C05373=1017.378,25.975,-122.265,-24.216,21.496,-42.540
C05374=1017.376,26.375,-122.301,-24.217,21.496,-42.534
C05375=1017.374,26.774,-122.336,-24.218,21.495,-42.529
C05376=1017.373,27.173,-122.371,-24.218,21.494,-42.525
C05377=1017.372,27.573,-122.406,-24.219,21.495,-42.520
C05378=1017.370,27.972,-122.441,-24.219,21.493,-42.516
C05379=1017.368,28.372,-122.475,-24.220,21.493,-42.510
C05380=1017.366,28.772,-122.511,-24.221,21.493,-42.507
C05381=1017.364,29.171,-122.546,-24.221,21.492,-42.501
C05382=1017.363,29.570,-122.580,-24.222,21.492,-42.497
C05383=1017.360,29.970,-122.616,-24.223,21.492,-42.492
C05384=1017.358,30.370,-122.650,-24.223,21.491,-42.488
C05385=1017.357,30.769,-122.685,-24.224,21.491,-42.483
C05386=1017.354,31.168,-122.721,-24.224,21.490,-42.479
C05387=1017.354,31.568,-122.756,-24.225,21.490,-42.474
C05388=1017.351,31.968,-122.791,-24.226,21.489,-42.469
C05389=1017.349,32.368,-122.826,-24.226,21.489,-42.464
C05390=1017.347,32.767,-122.861,-24.227,21.489,-42.461
C05391=1017.345,33.166,-122.896,-24.228,21.489,-42.455
C05392=1017.344,33.567,-122.932,-24.228,21.487,-42.451
C05393=1017.341,33.966,-122.968,-24.229,21.488,-42.446
C05394=1017.339,34.366,-123.002,-24.229,21.487,-42.442
C05395=1017.337,34.766,-123.037,-24.230,21.486,-42.437
C05396=1017.335,35.165,-123.073,-24.231,21.486,-42.433
C05397=1017.334,35.565,-123.108,-24.231,21.486,-42.428
C05398=1017.331,35.965,-123.143,-24.232,21.486,-42.424
C05399=1017.329,36.365,-123.178,-24.233,21.485,-42.418
C05400=1017.327,36.764,-123.214,-24.233,21.484,-42.414
C05401=1017.325,37.164,-123.250,-24.234,21.485,-42.409
C05402=1017.323,37.564,-123.284,-24.235,21.484,-42.405
C05403=1017.321,37.964,-123.320,-24.235,21.483,-42.400
C05404=1017.318,38.363,-123.355,-24.236,21.483,-42.396
C05405=1017.316,38.764,-123.391,-24.237,21.483,-42.391
C05406=1017.314,39.164,-123.426,-24.237,21.483,-42.387
C05407=1017.312,39.563,-123.461,-24.238,21.482,-42.383
C05408=1017.310,39.964,-123.497,-24.238,21.481,-42.378
C05409=1017.307,40.363,-123.533,-24.239,21.481,-42.374
C05410=1017.305,40.763,-123.568,-24.240,21.481,-42.369
C05411=1017.303,41.164,-123.603,-24.240,21.481,-42.365
C05412=1017.301,41.563,-123.639,-24.241,21.480,-42.359
C05413=1017.297,41.964,-123.674,-24.241,21.479,-42.356
C05414=1017.295,42.363,-123.710,-24.242,21.479,-42.352
C05415=1017.293,42.763,-123.746,-24.243,21.479,-42.347
C05416=1017.291,43.163,-123.781,-24.243,21.479,-42.343
C05417=1017.288,43.563,-123.816,-24.244,21.479,-42.338
C05418=1017.286,43.964,-123.853,-24.244,21.477,-42.333
C05419=1017.284,44.363,-123.888,-24.245,21.477,-42.330
C05420=1017.281,44.763,-123.924,-24.246,21.477,-42.325
C05421=1017.279,45.164,-123.959,-24.246,21.477,-42.321
C05422=1017.276,45.563,-123.995,-24.247,21.477,-42.316
C05423=1017.274,45.964,-124.031,-24.247,21.475,-42.311
C05424=1017.271,46.363,-124.067,-24.248,21.475,-42.308
C05425=1017.269,46.764,-124.102,-24.249,21.475,-42.302
C05426=1017.266,47.164,-124.138,-24.249,21.475,-42.299
C05427=1017.264,47.564,-124.174,-24.250,21.474,-42.295
C05428=1017.261,47.964,-124.210,-24.251,21.474,-42.290
C05429=1017.259,48.364,-124.245,-24.251,21.474,-42.286
C05430=1017.256,48.764,-124.281,-24.251,21.472,-42.282
C05431=1017.253,49.164,-124.317,-24.252,21.473,-42.277
C05432=1017.251,49.565,-124.353,-24.253,21.472,-42.273
C05433=1017.248,49.965,-124.389,-24.254,21.472,-42.268
C05434=1017.245,50.364,-124.424,-24.254,21.472,-42.264
C05435=1017.243,50.765,-124.461,-24.255,21.471,-42.260
C05436=1017.239,51.165,-124.496,-24.255,21.471,-42.255
C05437=1017.237,51.565,-124.532,-24.256,21.471,-42.251
C05438=1017.235,51.965,-124.568,-24.256,21.470,-42.247
C05439=1017.232,52.365,-124.604,-24.257,21.469,-42.243
C05440=1017.229,52.765,-124.640,-24.258,21.469,-42.238
C05441=1017.227,53.166,-124.675,-24.258,21.469,-42.234
C05442=1017.223,53.566,-124.712,-24.259,21.468,-42.230
C05443=1017.220,53.966,-124.748,-24.259,21.468,-42.225
C05444=1017.218,54.366,-124.784,-24.260,21.468,-42.221
C05445=1017.215,54.767,-124.820,-24.260,21.468,-42.218
C05446=1017.211,55.167,-124.856,-24.261,21.468,-42.212
C05447=1017.209,55.567,-124.892,-24.262,21.467,-42.209
C05448=1017.206,55.967,-124.928,-24.262,21.467,-42.205
C05449=1017.203,56.367,-124.964,-24.263,21.465,-42.201
C05450=1017.200,56.768,-125.000,-24.264,21.466,-42.196
C05451=1017.197,57.168,-125.036,-24.264,21.465,-42.192
C05452=1017.194,57.568,-125.072,-24.264,21.465,-42.188
C05453=1017.192,57.968,-125.109,-24.265,21.465,-42.183
C05454=1017.188,58.368,-125.145,-24.266,21.464,-42.179
C05455=1017.185,58.769,-125.180,-24.266,21.464,-42.175
C05456=1017.182,59.168,-125.217,-24.267,21.463,-42.172
C05457=1017.180,59.569,-125.253,-24.268,21.464,-42.166
C05458=1017.176,59.969,-125.289,-24.268,21.463,-42.163
C05459=1017.173,60.369,-125.325,-24.269,21.463,-42.159
C05460=1017.170,60.769,-125.361,-24.269,21.462,-42.155
C05461=1017.167,61.169,-125.399,-24.270,21.462,-42.150
C05462=1017.164,61.570,-125.434,-24.270,21.462,-42.146
C05463=1017.161,61.970,-125.470,-24.271,21.461,-42.142
C05464=1017.158,62.370,-125.506,-24.271,21.461,-42.139
C05465=1017.154,62.790,-125.545,-24.272,21.460,-42.133
C05466=1017.153,63.043,-125.568,-24.272,21.460,-42.131
C05467=1017.150,63.311,-125.593,-24.273,21.460,-42.129
C05468=1017.148,63.561,-125.615,-24.273,21.459,-42.127
C05469=1017.146,63.777,-125.634,-24.274,21.460,-42.124
C05470=1017.144,63.984,-125.653,-24.274,21.460,-42.122
C05471=1017.143,64.202,-125.673,-24.274,21.459,-42.120
C05472=1017.141,64.431,-125.693,-24.274,21.459,-42.116
C05473=1017.139,64.668,-125.715,-24.275,21.459,-42.115
C05474=1017.138,64.903,-125.737,-24.275,21.458,-42.113
C05475=1017.135,65.133,-125.758,-24.275,21.458,-42.111
C05476=1017.134,65.355,-125.778,-24.276,21.459,-42.108
C05477=1017.131,65.568,-125.797,-24.276,21.458,-42.106
C05478=1017.128,65.975,-125.834,-24.277,21.458,-42.102
C05479=1017.125,66.374,-125.870,-24.277,21.457,-42.098
C05480=1017.121,66.774,-125.907,-24.278,21.457,-42.094
C05481=1017.118,67.177,-125.943,-24.278,21.457,-42.089
C05482=1017.115,67.581,-125.980,-24.279,21.457,-42.085
C05483=1017.111,67.985,-126.017,-24.279,21.456,-42.082
C05484=1017.109,68.391,-126.053,-24.280,21.456,-42.078
C05485=1017.104,68.798,-126.091,-24.280,21.455,-42.074
C05486=1017.101,69.207,-126.128,-24.281,21.455,-42.069
C05487=1017.098,69.617,-126.166,-24.282,21.455,-42.065
C05488=1017.094,70.028,-126.204,-24.282,21.454,-42.061
C05489=1017.090,70.440,-126.241,-24.283,21.454,-42.058
C05490=1017.087,70.850,-126.278,-24.283,21.453,-42.054
C05491=1017.083,71.261,-126.316,-24.284,21.454,-42.049
C05492=1017.079,71.673,-126.353,-24.285,21.453,-42.045
C05493=1017.076,72.084,-126.391,-24.285,21.453,-42.041
C05494=1017.072,72.498,-126.429,-24.285,21.452,-42.037
C05495=1017.069,72.913,-126.467,-24.286,21.452,-42.034
C05496=1017.064,73.331,-126.505,-24.287,21.452,-42.028
C05497=1017.061,73.752,-126.543,-24.287,21.452,-42.025
C05498=1017.059,73.963,-126.563,-24.288,21.451,-42.023
C05499=1017.057,74.175,-126.582,-24.288,21.451,-42.021
C05500=1017.055,74.388,-126.602,-24.288,21.451,-42.019
C05501=1017.054,74.601,-126.621,-24.288,21.451,-42.017
C05502=1017.051,74.815,-126.641,-24.289,21.450,-42.015
C05503=1017.050,75.028,-126.660,-24.289,21.451,-42.012
C05504=1017.047,75.242,-126.680,-24.289,21.451,-42.010
C05505=1017.045,75.454,-126.699,-24.290,21.450,-42.008
C05506=1017.041,75.873,-126.738,-24.290,21.450,-42.004
C05507=1017.037,76.286,-126.776,-24.291,21.449,-42.001
C05508=1017.034,76.687,-126.812,-24.291,21.449,-41.997
C05509=1017.030,77.082,-126.848,-24.292,21.449,-41.994
C05510=1017.026,77.471,-126.885,-24.292,21.448,-41.989
C05511=1017.023,77.856,-126.919,-24.293,21.447,-41.986
C05512=1017.019,78.243,-126.954,-24.293,21.448,-41.980
C05513=1017.015,78.634,-126.991,-24.294,21.447,-41.977
C05514=1017.011,79.031,-127.028,-24.294,21.447,-41.973
C05515=1017.008,79.436,-127.065,-24.295,21.447,-41.970
C05516=1017.004,79.850,-127.103,-24.296,21.447,-41.966
C05517=1017.001,80.061,-127.122,-24.296,21.446,-41.964
C05518=1016.999,80.273,-127.141,-24.296,21.446,-41.962
C05519=1016.997,80.485,-127.161,-24.296,21.446,-41.960
C05520=1016.995,80.698,-127.180,-24.297,21.446,-41.958
C05521=1016.993,80.911,-127.200,-24.297,21.445,-41.956
C05522=1016.991,81.124,-127.220,-24.297,21.445,-41.955
C05523=1016.989,81.336,-127.239,-24.297,21.445,-41.953
C05524=1016.986,81.549,-127.259,-24.298,21.445,-41.951
C05525=1016.984,81.760,-127.278,-24.298,21.445,-41.949
C05526=1016.982,81.972,-127.298,-24.298,21.444,-41.947
C05527=1016.980,82.184,-127.317,-24.299,21.445,-41.944
C05528=1016.979,82.395,-127.337,-24.299,21.444,-41.942
C05529=1016.976,82.606,-127.356,-24.299,21.444,-41.940
C05530=1016.973,82.816,-127.376,-24.299,21.444,-41.938
C05531=1016.970,83.236,-127.414,-24.300,21.444,-41.935
C05532=1016.965,83.656,-127.453,-24.300,21.444,-41.931
C05533=1016.961,84.072,-127.492,-24.301,21.443,-41.927
C05534=1016.957,84.488,-127.530,-24.301,21.443,-41.923
C05535=1016.953,84.902,-127.568,-24.302,21.443,-41.920
C05536=1016.949,85.315,-127.606,-24.302,21.442,-41.916
C05537=1016.944,85.726,-127.644,-24.303,21.442,-41.912
C05538=1016.940,86.135,-127.682,-24.303,21.441,-41.908
C05539=1016.935,86.542,-127.719,-24.304,21.442,-41.905
C05540=1016.931,86.948,-127.756,-24.304,21.441,-41.901
C05541=1016.927,87.350,-127.794,-24.305,21.441,-41.898
C05542=1016.923,87.747,-127.831,-24.305,21.440,-41.894
C05543=1016.919,88.135,-127.867,-24.306,21.440,-41.890
C05544=1016.914,88.518,-127.902,-24.307,21.440,-41.887
C05545=1016.910,88.901,-127.937,-24.307,21.440,-41.883
C05546=1016.907,89.288,-127.973,-24.308,21.439,-41.879
C05547=1016.903,89.681,-128.010,-24.308,21.439,-41.875
C05548=1016.898,90.079,-128.046,-24.309,21.439,-41.872
C05549=1016.894,90.478,-128.083,-24.309,21.439,-41.868
C05550=1016.890,90.877,-128.120,-24.310,21.438,-41.865
C05551=1016.884,91.277,-128.157,-24.310,21.438,-41.861
C05552=1016.880,91.675,-128.194,-24.311,21.438,-41.857
C05553=1016.876,92.074,-128.231,-24.311,21.438,-41.854
C05554=1016.872,92.474,-128.268,-24.312,21.437,-41.850
C05555=1016.867,92.873,-128.305,-24.312,21.437,-41.846
C05556=1016.863,93.272,-128.342,-24.312,21.437,-41.844
C05557=1016.859,93.671,-128.379,-24.313,21.436,-41.841
C05558=1016.854,94.070,-128.416,-24.313,21.436,-41.837
C05559=1016.850,94.469,-128.454,-24.314,21.435,-41.833
C05560=1016.845,94.867,-128.490,-24.315,21.436,-41.830
C05561=1016.840,95.266,-128.528,-24.315,21.435,-41.826
C05562=1016.836,95.666,-128.564,-24.316,21.435,-41.822
C05563=1016.832,96.065,-128.601,-24.316,21.435,-41.819
C05564=1016.827,96.464,-128.639,-24.317,21.435,-41.815
C05565=1016.822,96.862,-128.676,-24.317,21.434,-41.811
C05566=1016.817,97.261,-128.713,-24.318,21.434,-41.808
C05567=1016.813,97.660,-128.750,-24.318,21.433,-41.806
C05568=1016.809,98.059,-128.787,-24.318,21.433,-41.802
C05569=1016.803,98.458,-128.824,-24.319,21.432,-41.798
C05570=1016.799,98.856,-128.861,-24.319,21.433,-41.795
C05571=1016.794,99.256,-128.899,-24.320,21.432,-41.791
C05572=1016.790,99.654,-128.935,-24.320,21.432,-41.787
C05573=1016.785,100.053,-128.973,-24.321,21.432,-41.784
C05574=1016.780,100.452,-129.009,-24.322,21.432,-41.780
C05575=1016.775,100.851,-129.047,-24.322,21.431,-41.778
C05576=1016.770,101.249,-129.083,-24.322,21.431,-41.775
C05577=1016.765,101.648,-129.121,-24.323,21.431,-41.771
C05578=1016.761,102.047,-129.159,-24.323,21.430,-41.767
C05579=1016.756,102.445,-129.195,-24.324,21.430,-41.763
C05580=1016.751,102.844,-129.233,-24.324,21.430,-41.760
C05581=1016.746,103.242,-129.270,-24.325,21.430,-41.756
C05582=1016.741,103.641,-129.307,-24.325,21.430,-41.754
C05583=1016.736,104.040,-129.345,-24.326,21.429,-41.751
C05584=1016.731,104.438,-129.381,-24.326,21.429,-41.747
C05585=1016.727,104.837,-129.419,-24.327,21.429,-41.743
C05586=1016.721,105.236,-129.456,-24.327,21.429,-41.740
C05587=1016.717,105.635,-129.493,-24.328,21.428,-41.736
C05588=1016.712,106.033,-129.531,-24.328,21.428,-41.734
C05589=1016.706,106.431,-129.568,-24.328,21.427,-41.730
C05590=1016.701,106.831,-129.606,-24.329,21.427,-41.727
C05591=1016.697,107.229,-129.642,-24.330,21.427,-41.723
C05592=1016.691,107.627,-129.680,-24.330,21.427,-41.719
C05593=1016.686,108.026,-129.717,-24.330,21.426,-41.717
C05594=1016.681,108.425,-129.755,-24.331,21.426,-41.714
C05595=1016.676,108.823,-129.791,-24.331,21.426,-41.710
C05596=1016.671,109.221,-129.829,-24.332,21.426,-41.707
C05597=1016.666,109.620,-129.866,-24.332,21.426,-41.703
C05598=1016.661,110.019,-129.904,-24.333,21.425,-41.701
C05599=1016.655,110.417,-129.941,-24.333,21.425,-41.697
C05600=1016.650,110.816,-129.978,-24.334,21.425,-41.694
C05601=1016.645,111.215,-130.016,-24.334,21.425,-41.690
C05602=1016.639,111.613,-130.053,-24.334,21.424,-41.688
C05603=1016.634,112.012,-130.090,-24.335,21.423,-41.684
C05604=1016.629,112.410,-130.128,-24.335,21.424,-41.681
C05605=1016.624,112.808,-130.164,-24.336,21.423,-41.677
C05606=1016.618,113.207,-130.202,-24.336,21.423,-41.675
C05607=1016.614,113.606,-130.239,-24.337,21.423,-41.671
C05608=1016.608,114.004,-130.277,-24.337,21.422,-41.668
C05609=1016.602,114.403,-130.315,-24.338,21.423,-41.664
C05610=1016.597,114.801,-130.352,-24.338,21.422,-41.662
C05611=1016.591,115.200,-130.389,-24.339,21.422,-41.659
C05612=1016.586,115.598,-130.426,-24.339,21.422,-41.655
C05613=1016.580,115.997,-130.464,-24.340,21.422,-41.652
C05614=1016.575,116.395,-130.501,-24.340,21.421,-41.649
C05615=1016.570,116.787,-130.539,-24.340,21.420,-41.646
C05616=1016.564,117.192,-130.576,-24.341,21.421,-41.642
C05617=1016.559,117.590,-130.613,-24.341,21.420,-41.638
C05618=1016.552,117.989,-130.651,-24.342,21.420,-41.637
C05619=1016.547,118.387,-130.688,-24.342,21.420,-41.633
C05620=1016.541,118.786,-130.725,-24.343,21.420,-41.629
C05621=1016.536,119.184,-130.763,-24.343,21.420,-41.626
C05622=1016.531,119.582,-130.801,-24.343,21.419,-41.624
C05623=1016.525,119.981,-130.839,-24.344,21.419,-41.620
C05624=1016.519,120.379,-130.876,-24.345,21.419,-41.617
C05625=1016.514,120.778,-130.913,-24.345,21.418,-41.614
C05626=1016.509,121.177,-130.951,-24.345,21.418,-41.611
C05627=1016.503,121.575,-130.989,-24.346,21.418,-41.607
C05628=1016.498,121.973,-131.027,-24.346,21.417,-41.605
C05629=1016.493,122.373,-131.064,-24.347,21.418,-41.602
C05630=1016.487,122.771,-131.102,-24.347,21.417,-41.598
C05631=1016.482,123.169,-131.140,-24.348,21.418,-41.595
C05632=1016.476,123.568,-131.178,-24.348,21.416,-41.592
C05633=1016.471,123.967,-131.215,-24.348,21.417,-41.589
C05634=1016.465,124.365,-131.254,-24.349,21.416,-41.585
C05635=1016.460,124.763,-131.291,-24.349,21.416,-41.583
C05636=1016.455,125.162,-131.328,-24.350,21.416,-41.580
C05637=1016.449,125.560,-131.367,-24.350,21.416,-41.576
C05638=1016.444,125.959,-131.405,-24.350,21.415,-41.574
C05639=1016.438,126.357,-131.442,-24.351,21.415,-41.571
C05640=1016.432,126.756,-131.480,-24.351,21.415,-41.567
C05641=1016.427,127.154,-131.518,-24.352,21.415,-41.565
C05642=1016.422,127.553,-131.556,-24.352,21.414,-41.561
C05643=1016.416,127.952,-131.593,-24.353,21.415,-41.558
C05644=1016.410,128.350,-131.631,-24.353,21.414,-41.555
C05645=1016.405,128.748,-131.669,-24.354,21.414,-41.552
C05646=1016.399,129.147,-131.707,-24.354,21.413,-41.550
C05647=1016.393,129.546,-131.745,-24.354,21.413,-41.547
C05648=1016.388,129.945,-131.783,-24.355,21.413,-41.543
C05649=1016.382,130.343,-131.821,-24.355,21.413,-41.541
C05650=1016.376,130.741,-131.859,-24.356,21.413,-41.538
C05651=1016.370,131.140,-131.896,-24.356,21.413,-41.534
C05652=1016.364,131.539,-131.934,-24.356,21.412,-41.532
C05653=1016.359,131.938,-131.972,-24.357,21.412,-41.528
C05654=1016.353,132.336,-132.011,-24.357,21.412,-41.525
C05655=1016.347,132.735,-132.048,-24.358,21.411,-41.523
C05656=1016.341,133.134,-132.086,-24.358,21.412,-41.519
C05657=1016.336,133.532,-132.124,-24.358,21.411,-41.517
C05658=1016.329,133.931,-132.162,-24.359,21.411,-41.514
C05659=1016.323,134.329,-132.200,-24.359,21.411,-41.510
C05660=1016.318,134.728,-132.238,-24.360,21.410,-41.508
C05661=1016.312,135.127,-132.276,-24.360,21.411,-41.505
C05662=1016.306,135.522,-132.313,-24.360,21.410,-41.502
C05663=1016.300,135.894,-132.349,-24.361,21.409,-41.500
C05664=1016.295,136.233,-132.381,-24.361,21.410,-41.497
C05665=1016.290,136.551,-132.412,-24.361,21.409,-41.495
C05666=1016.285,136.867,-132.441,-24.362,21.409,-41.491
C05667=1016.281,137.204,-132.474,-24.363,21.410,-41.488
C05668=1016.275,137.573,-132.509,-24.363,21.408,-41.486
C05669=1016.269,137.974,-132.547,-24.363,21.408,-41.484
C05670=1016.266,138.180,-132.567,-24.363,21.408,-41.482
C05671=1016.262,138.398,-132.587,-24.364,21.408,-41.480
C05672=1016.259,138.634,-132.610,-24.364,21.408,-41.478
C05673=1016.255,138.895,-132.635,-24.364,21.407,-41.476
C05674=1016.250,139.172,-132.661,-24.364,21.408,-41.475
C05675=1016.246,139.460,-132.689,-24.365,21.408,-41.473
C05676=1016.242,139.747,-132.716,-24.365,21.408,-41.471
C05677=1016.237,140.024,-132.743,-24.365,21.408,-41.470
C05678=1016.233,140.283,-132.767,-24.366,21.408,-41.468
C05679=1016.230,140.519,-132.790,-24.366,21.408,-41.466
C05680=1016.223,140.937,-132.830,-24.366,21.407,-41.462
C05681=1016.217,141.341,-132.868,-24.366,21.406,-41.460
C05682=1016.211,141.746,-132.907,-24.367,21.407,-41.457
C05683=1016.204,142.153,-132.945,-24.368,21.406,-41.453
C05684=1016.198,142.559,-132.984,-24.368,21.406,-41.451
C05685=1016.191,142.967,-133.024,-24.368,21.406,-41.448
C05686=1016.184,143.376,-133.062,-24.369,21.405,-41.445
C05687=1016.178,143.785,-133.101,-24.369,21.406,-41.442
C05688=1016.171,144.195,-133.140,-24.370,21.405,-41.438
C05689=1016.165,144.606,-133.180,-24.370,21.405,-41.436
C05690=1016.159,145.018,-133.219,-24.370,21.405,-41.432
C05691=1016.152,145.430,-133.258,-24.371,21.404,-41.431
C05692=1016.145,145.842,-133.298,-24.371,21.405,-41.427
C05693=1016.139,146.256,-133.337,-24.372,21.404,-41.424
C05694=1016.131,146.668,-133.377,-24.372,21.404,-41.422
C05695=1016.125,147.082,-133.416,-24.372,21.404,-41.418
C05696=1016.118,147.496,-133.456,-24.373,21.403,-41.416
C05697=1016.112,147.909,-133.495,-24.373,21.403,-41.412
C05698=1016.105,148.324,-133.535,-24.374,21.403,-41.409
C05699=1016.098,148.738,-133.574,-24.374,21.403,-41.407
C05700=1016.091,149.151,-133.614,-24.375,21.403,-41.403
C05701=1016.084,149.566,-133.653,-24.375,21.402,-41.401
C05702=1016.077,149.979,-133.693,-24.375,21.402,-41.398
C05703=1016.070,150.394,-133.732,-24.376,21.402,-41.394
C05704=1016.063,150.806,-133.772,-24.376,21.401,-41.392
C05705=1016.056,151.220,-133.811,-24.377,21.402,-41.389
C05706=1016.049,151.634,-133.851,-24.377,21.402,-41.387
C05707=1016.042,152.047,-133.891,-24.377,21.401,-41.383
C05708=1016.035,152.460,-133.930,-24.378,21.401,-41.381
C05709=1016.028,152.871,-133.969,-24.378,21.400,-41.377
C05710=1016.021,153.284,-134.009,-24.378,21.400,-41.375
C05711=1016.015,153.695,-134.048,-24.379,21.401,-41.372
C05712=1016.007,154.105,-134.087,-24.380,21.400,-41.368
C05713=1016.000,154.515,-134.127,-24.380,21.400,-41.366
C05714=1015.993,154.924,-134.165,-24.380,21.400,-41.363
C05715=1015.986,155.332,-134.205,-24.381,21.399,-41.361
C05716=1015.979,155.740,-134.244,-24.381,21.400,-41.358
C05717=1015.971,156.147,-134.283,-24.381,21.399,-41.355
C05718=1015.964,156.552,-134.321,-24.382,21.399,-41.352
C05719=1015.957,156.958,-134.360,-24.382,21.399,-41.350
C05720=1015.949,157.362,-134.399,-24.383,21.398,-41.346
C05721=1015.943,157.766,-134.437,-24.383,21.398,-41.344
C05722=1015.936,158.168,-134.476,-24.383,21.399,-41.341
C05723=1015.928,158.570,-134.514,-24.384,21.397,-41.339
C05724=1015.922,158.971,-134.553,-24.384,21.398,-41.335
C05725=1015.914,159.372,-134.592,-24.384,21.398,-41.333
C05726=1015.908,159.772,-134.630,-24.385,21.397,-41.330
C05727=1015.907,160.169,-134.672,-24.385,21.397,-41.328
C05728=1015.905,160.573,-134.714,-24.386,21.397,-41.325
C05729=1015.904,160.787,-134.736,-24.386,21.397,-41.324
C05730=1015.903,161.011,-134.760,-24.386,21.396,-41.322
C05731=1015.902,161.248,-134.784,-24.386,21.396,-41.320
C05732=1015.901,161.499,-134.811,-24.387,21.397,-41.319
C05733=1015.900,161.762,-134.838,-24.387,21.397,-41.317
C05734=1015.900,162.032,-134.866,-24.387,21.396,-41.315
C05735=1015.898,162.303,-134.895,-24.387,21.396,-41.313
C05736=1015.897,162.572,-134.923,-24.388,21.396,-41.311
C05737=1015.897,162.835,-134.950,-24.388,21.396,-41.309
C05738=1015.896,163.089,-134.978,-24.388,21.395,-41.308
C05739=1015.895,163.324,-135.003,-24.388,21.396,-41.306
C05740=1015.894,163.736,-135.045,-24.389,21.395,-41.304
C05741=1015.892,163.926,-135.065,-24.389,21.395,-41.302
C05742=1015.891,164.312,-135.106,-24.389,21.395,-41.300
C05743=1015.890,164.712,-135.147,-24.390,21.395,-41.297
C05744=1015.888,165.113,-135.190,-24.390,21.395,-41.295
C05745=1015.887,165.513,-135.232,-24.390,21.394,-41.291
C05746=1015.885,165.913,-135.274,-24.391,21.394,-41.289
C05747=1015.884,166.313,-135.316,-24.391,21.395,-41.286
C05748=1015.883,166.714,-135.359,-24.391,21.393,-41.284
C05749=1015.881,167.114,-135.400,-24.392,21.394,-41.280
C05750=1015.880,167.514,-135.443,-24.392,21.394,-41.278
C05751=1015.878,167.916,-135.485,-24.393,21.394,-41.275
C05752=1015.877,168.315,-135.527,-24.393,21.393,-41.273
C05753=1015.875,168.716,-135.569,-24.393,21.393,-41.271
C05754=1015.875,169.116,-135.612,-24.394,21.393,-41.267
C05755=1015.872,169.517,-135.654,-24.394,21.392,-41.265
C05756=1015.871,169.917,-135.697,-24.395,21.392,-41.262
C05757=1015.870,170.318,-135.738,-24.395,21.392,-41.260
C05758=1015.869,170.719,-135.781,-24.395,21.392,-41.256
C05759=1015.866,171.119,-135.823,-24.396,21.392,-41.254
C05760=1015.866,171.519,-135.865,-24.396,21.392,-41.251
C05761=1015.864,171.920,-135.908,-24.396,21.392,-41.249
C05762=1015.863,172.321,-135.950,-24.397,21.391,-41.247
C05763=1015.862,172.721,-135.993,-24.397,21.391,-41.243
C05764=1015.861,173.122,-136.035,-24.397,21.391,-41.242
C05765=1015.859,173.523,-136.078,-24.398,21.390,-41.238
C05766=1015.858,173.924,-136.120,-24.398,21.390,-41.236
C05767=1015.857,174.324,-136.163,-24.399,21.391,-41.233
C05768=1015.856,174.725,-136.206,-24.399,21.390,-41.231
C05769=1015.854,175.126,-136.248,-24.400,21.390,-41.227
C05770=1015.853,175.526,-136.291,-24.400,21.390,-41.225
C05771=1015.851,175.927,-136.333,-24.400,21.390,-41.223
C05772=1015.850,176.328,-136.376,-24.401,21.389,-41.219
C05773=1015.849,176.728,-136.418,-24.401,21.389,-41.218
C05774=1015.847,177.129,-136.461,-24.401,21.389,-41.214
C05775=1015.846,177.530,-136.503,-24.402,21.389,-41.212
C05776=1015.845,177.930,-136.546,-24.402,21.389,-41.209
C05777=1015.844,178.332,-136.589,-24.402,21.388,-41.207
C05778=1015.842,178.732,-136.632,-24.403,21.388,-41.205
C05779=1015.841,179.133,-136.675,-24.403,21.388,-41.201
C05780=1015.840,179.533,-136.718,-24.403,21.388,-41.199
C05781=1015.838,179.935,-136.760,-24.404,21.388,-41.196
C05782=1015.838,180.336,-136.803,-24.404,21.388,-41.194
C05783=1015.837,180.736,-136.846,-24.405,21.387,-41.190
C05784=1015.835,181.137,-136.889,-24.405,21.387,-41.188
C05785=1015.834,181.538,-136.931,-24.405,21.387,-41.186
C05786=1015.833,181.939,-136.974,-24.406,21.387,-41.183
C05787=1015.832,182.340,-137.018,-24.406,21.386,-41.181
C05788=1015.831,182.741,-137.061,-24.407,21.387,-41.177
C05789=1015.829,183.142,-137.103,-24.407,21.386,-41.176
C05790=1015.828,183.543,-137.146,-24.407,21.386,-41.172
C05791=1015.827,183.943,-137.189,-24.408,21.386,-41.170
C05792=1015.826,184.345,-137.232,-24.408,21.386,-41.168
C05793=1015.825,184.745,-137.275,-24.409,21.386,-41.165
C05794=1015.824,185.146,-137.319,-24.409,21.385,-41.162
C05795=1015.822,185.547,-137.362,-24.409,21.385,-41.159
C05796=1015.821,185.949,-137.405,-24.410,21.385,-41.157
C05797=1015.820,186.350,-137.448,-24.410,21.384,-41.155
C05798=1015.819,186.751,-137.491,-24.410,21.384,-41.151
C05799=1015.818,187.152,-137.534,-24.411,21.384,-41.150
C05800=1015.817,187.552,-137.577,-24.411,21.385,-41.146
C05801=1015.816,187.954,-137.621,-24.411,21.384,-41.144
C05802=1015.815,188.355,-137.664,-24.412,21.384,-41.141
C05803=1015.814,188.755,-137.707,-24.412,21.384,-41.139
C05804=1015.813,189.157,-137.750,-24.412,21.384,-41.137
C05805=1015.812,189.558,-137.794,-24.413,21.383,-41.133
C05806=1015.810,189.959,-137.837,-24.413,21.383,-41.131
C05807=1015.810,190.360,-137.880,-24.414,21.383,-41.128
C05808=1015.809,190.761,-137.924,-24.414,21.383,-41.126
C05809=1015.808,191.162,-137.967,-24.414,21.382,-41.124
C05810=1015.807,191.564,-138.010,-24.415,21.382,-41.120
C05811=1015.806,191.964,-138.055,-24.415,21.382,-41.118
C05812=1015.805,192.365,-138.098,-24.415,21.382,-41.115
C05813=1015.804,192.766,-138.141,-24.416,21.382,-41.113
C05814=1015.803,193.167,-138.184,-24.416,21.382,-41.109
C05815=1015.803,193.569,-138.228,-24.417,21.382,-41.108
C05816=1015.801,193.970,-138.272,-24.417,21.381,-41.105
C05817=1015.801,194.371,-138.316,-24.417,21.381,-41.102
C05818=1015.800,194.772,-138.359,-24.418,21.381,-41.100
C05819=1015.799,195.173,-138.402,-24.418,21.381,-41.097
C05820=1015.798,195.575,-138.446,-24.418,21.380,-41.094
C05821=1015.797,195.976,-138.490,-24.419,21.381,-41.091
C05822=1015.796,196.376,-138.534,-24.419,21.380,-41.089
C05823=1015.796,196.778,-138.577,-24.419,21.380,-41.087
C05824=1015.794,197.179,-138.621,-24.420,21.380,-41.084
C05825=1015.794,197.580,-138.665,-24.420,21.380,-41.082
C05826=1015.793,197.981,-138.708,-24.421,21.380,-41.078
C05827=1015.792,198.382,-138.751,-24.421,21.379,-41.076
C05828=1015.791,198.783,-138.796,-24.421,21.379,-41.074
C05829=1015.790,199.181,-138.840,-24.422,21.379,-41.071
C05830=1015.789,199.571,-138.882,-24.422,21.379,-41.069
C05831=1015.789,199.971,-138.926,-24.423,21.378,-41.065
C05832=1015.789,200.184,-138.949,-24.423,21.378,-41.065
C05833=1015.788,200.407,-138.973,-24.423,21.378,-41.063
C05834=1015.788,200.636,-138.998,-24.423,21.378,-41.061
C05835=1015.787,200.863,-139.023,-24.423,21.379,-41.060
C05836=1015.787,201.270,-139.067,-24.424,21.378,-41.058
C05837=1015.786,201.622,-139.106,-24.424,21.378,-41.054
C05838=1015.785,201.971,-139.144,-24.424,21.378,-41.052
C05839=1015.787,202.358,-139.188,-24.425,21.378,-41.051
C05840=1015.792,203.574,-139.323,-24.373,21.403,-41.416
C05841=1015.794,203.823,-139.350,-24.373,21.404,-41.415
C05842=1015.795,204.071,-139.379,-24.373,21.403,-41.414
C05843=1015.797,204.320,-139.406,-24.373,21.403,-41.412
C05844=1015.800,204.568,-139.433,-24.374,21.404,-41.411
C05845=1015.801,204.817,-139.460,-24.373,21.403,-41.410
C05846=1015.803,205.066,-139.487,-24.374,21.403,-41.409
C05847=1015.805,205.314,-139.516,-24.374,21.403,-41.407
C05848=1015.807,205.562,-139.543,-24.374,21.402,-41.407
C05849=1015.809,205.811,-139.570,-24.374,21.403,-41.405
C05850=1015.810,206.059,-139.598,-24.375,21.403,-41.403
C05851=1015.812,206.307,-139.625,-24.375,21.402,-41.401
C05852=1015.814,206.556,-139.652,-24.375,21.402,-41.401
C05853=1015.816,206.805,-139.679,-24.375,21.402,-41.399
C05854=1015.818,207.053,-139.707,-24.375,21.402,-41.398
C05855=1015.819,207.301,-139.735,-24.375,21.402,-41.398
C05856=1015.821,207.550,-139.762,-24.376,21.402,-41.396
C05857=1015.823,207.798,-139.790,-24.376,21.402,-41.394
C05858=1015.825,208.047,-139.817,-24.376,21.402,-41.392
C05859=1015.827,208.289,-139.844,-24.376,21.401,-41.392
C05860=1015.829,208.532,-139.871,-24.376,21.402,-41.391
C05861=1015.830,208.774,-139.898,-24.377,21.402,-41.389
C05862=1015.833,209.018,-139.924,-24.377,21.401,-41.388
C05863=1015.835,209.260,-139.952,-24.377,21.402,-41.387
C05864=1015.837,209.503,-139.978,-24.377,21.401,-41.385
C05865=1015.838,209.745,-140.006,-24.377,21.401,-41.383
C05866=1015.840,209.988,-140.033,-24.377,21.401,-41.383
C05867=1015.842,210.236,-140.060,-24.378,21.401,-41.381
C05868=1015.844,210.485,-140.087,-24.378,21.401,-41.379
C05869=1015.846,210.733,-140.115,-24.378,21.401,-41.378
C05870=1015.849,210.982,-140.142,-24.378,21.400,-41.377
C05871=1015.850,211.231,-140.171,-24.378,21.400,-41.375
C05872=1015.852,211.479,-140.198,-24.379,21.401,-41.374
C05873=1015.854,211.727,-140.226,-24.379,21.401,-41.372
C05874=1015.856,211.976,-140.253,-24.379,21.400,-41.372
C05875=1015.858,212.224,-140.281,-24.379,21.400,-41.370
C05876=1015.860,212.473,-140.309,-24.380,21.400,-41.368
C05877=1015.863,212.721,-140.336,-24.380,21.400,-41.366
C05878=1015.865,212.970,-140.363,-24.380,21.400,-41.366
C05879=1015.866,213.218,-140.392,-24.380,21.400,-41.365
C05880=1015.869,213.467,-140.419,-24.380,21.400,-41.363
C05881=1015.871,213.715,-140.447,-24.381,21.400,-41.361
C05882=1015.873,213.963,-140.475,-24.381,21.400,-41.359
C05883=1015.875,214.212,-140.502,-24.381,21.399,-41.359
C05884=1015.877,214.460,-140.530,-24.381,21.399,-41.357
C05885=1015.879,214.709,-140.557,-24.381,21.400,-41.356
C05886=1015.881,214.957,-140.586,-24.382,21.399,-41.354
C05887=1015.883,215.200,-140.613,-24.382,21.398,-41.353
C05888=1015.885,215.443,-140.639,-24.382,21.399,-41.352
C05889=1015.888,215.685,-140.667,-24.382,21.399,-41.350
C05890=1015.889,215.928,-140.694,-24.382,21.399,-41.348
C05891=1015.892,216.171,-140.722,-24.383,21.398,-41.346
C05892=1015.894,216.414,-140.748,-24.383,21.398,-41.346
C05893=1015.896,216.656,-140.775,-24.383,21.398,-41.344
C05894=1015.898,216.899,-140.803,-24.383,21.398,-41.342
C05895=1015.900,217.147,-140.831,-24.383,21.399,-41.341
C05896=1015.903,217.396,-140.858,-24.384,21.398,-41.339
C05897=1015.904,217.645,-140.886,-24.384,21.397,-41.339
C05898=1015.907,217.892,-140.914,-24.384,21.397,-41.337
C05899=1015.909,218.142,-140.942,-24.384,21.398,-41.335
C05900=1015.911,218.390,-140.970,-24.384,21.398,-41.333
C05901=1015.913,218.638,-140.997,-24.385,21.397,-41.332
C05902=1015.916,218.887,-141.026,-24.385,21.397,-41.330
C05903=1015.918,219.135,-141.053,-24.385,21.397,-41.330
C05904=1015.919,219.383,-141.081,-24.385,21.397,-41.328
C05905=1015.922,219.632,-141.109,-24.385,21.397,-41.326
C05906=1015.925,219.880,-141.137,-24.386,21.397,-41.324
C05907=1015.927,220.129,-141.166,-24.386,21.397,-41.323
C05908=1015.929,220.377,-141.193,-24.386,21.397,-41.321
C05909=1015.931,220.626,-141.221,-24.386,21.396,-41.320
C05910=1015.933,220.874,-141.249,-24.386,21.396,-41.318
C05911=1015.936,221.122,-141.277,-24.387,21.397,-41.317
C05912=1015.938,221.371,-141.306,-24.387,21.396,-41.315
C05913=1015.940,221.619,-141.333,-24.387,21.396,-41.313
C05914=1015.943,221.868,-141.362,-24.388,21.396,-41.311
C05915=1015.945,222.111,-141.388,-24.388,21.397,-41.310
C05916=1015.947,222.353,-141.416,-24.388,21.396,-41.309
C05917=1015.950,222.597,-141.443,-24.388,21.395,-41.308
C05918=1015.952,222.839,-141.471,-24.388,21.395,-41.306
C05919=1015.954,223.082,-141.498,-24.389,21.396,-41.304
C05920=1015.956,223.324,-141.525,-24.389,21.396,-41.302
C05921=1015.959,223.568,-141.553,-24.389,21.395,-41.300
C05922=1015.961,223.810,-141.581,-24.389,21.395,-41.300
C05923=1015.963,224.058,-141.608,-24.389,21.394,-41.298
C05924=1015.965,224.307,-141.637,-24.390,21.395,-41.297
C05925=1015.968,224.556,-141.665,-24.390,21.395,-41.295
C05926=1015.970,224.804,-141.693,-24.390,21.395,-41.293
C05927=1015.973,225.053,-141.721,-24.390,21.394,-41.291
C05928=1015.975,225.301,-141.749,-24.391,21.394,-41.289
C05929=1015.978,225.549,-141.778,-24.391,21.395,-41.288
C05930=1015.980,225.797,-141.805,-24.391,21.395,-41.286
C05931=1015.982,226.046,-141.834,-24.391,21.394,-41.285
C05932=1015.985,226.294,-141.862,-24.391,21.393,-41.284
C05933=1015.987,226.543,-141.890,-24.392,21.393,-41.282
C05934=1015.990,226.792,-141.919,-24.392,21.394,-41.280
C05935=1015.992,227.039,-141.946,-24.392,21.394,-41.278
C05936=1015.994,227.288,-141.975,-24.393,21.393,-41.276
C05937=1015.998,227.536,-142.004,-24.393,21.393,-41.275
C05938=1016.000,227.784,-142.031,-24.393,21.393,-41.273
C05939=1016.002,228.033,-142.060,-24.393,21.394,-41.271
C05940=1016.005,228.282,-142.088,-24.394,21.393,-41.269
C05941=1016.007,228.530,-142.116,-24.394,21.393,-41.267
C05942=1016.010,228.779,-142.144,-24.394,21.393,-41.266
C05943=1016.012,229.021,-142.172,-24.394,21.392,-41.265
C05944=1016.014,229.265,-142.200,-24.394,21.392,-41.263
C05945=1016.017,229.507,-142.228,-24.395,21.392,-41.262
C05946=1016.019,229.750,-142.256,-24.395,21.392,-41.260
C05947=1016.022,229.993,-142.283,-24.395,21.392,-41.258
C05948=1016.024,230.236,-142.311,-24.395,21.392,-41.256
C05949=1016.027,230.479,-142.339,-24.396,21.392,-41.254
C05950=1016.029,230.722,-142.366,-24.396,21.391,-41.252
C05951=1016.032,230.970,-142.395,-24.396,21.392,-41.251
C05952=1016.035,231.219,-142.423,-24.396,21.392,-41.249
C05953=1016.037,231.467,-142.451,-24.397,21.392,-41.247
C05954=1016.039,231.716,-142.480,-24.397,21.391,-41.245
C05955=1016.042,231.964,-142.509,-24.397,21.391,-41.243
C05956=1016.045,232.212,-142.537,-24.397,21.391,-41.242
C05957=1016.048,232.461,-142.565,-24.398,21.391,-41.240
C05958=1016.050,232.708,-142.594,-24.398,21.390,-41.238
C05959=1016.052,232.957,-142.622,-24.398,21.391,-41.236
C05960=1016.055,233.206,-142.650,-24.399,21.391,-41.234
C05961=1016.059,233.454,-142.679,-24.399,21.391,-41.233
C05962=1016.061,233.703,-142.708,-24.399,21.390,-41.231
C05963=1016.063,233.951,-142.736,-24.399,21.390,-41.229
C05964=1016.066,234.199,-142.765,-24.400,21.390,-41.227
C05965=1016.069,234.447,-142.793,-24.400,21.390,-41.225
C05966=1016.071,234.696,-142.822,-24.400,21.390,-41.223
C05967=1016.075,235.002,-142.857,-24.400,21.389,-41.221
C05968=1016.078,235.308,-142.892,-24.401,21.389,-41.219
C05969=1016.081,235.614,-142.927,-24.401,21.390,-41.216
C05970=1016.084,235.919,-142.963,-24.401,21.389,-41.214
C05971=1016.087,236.133,-142.987,-24.402,21.389,-41.212
C05972=1016.089,236.347,-143.012,-24.402,21.389,-41.210
C05973=1016.091,236.562,-143.036,-24.402,21.389,-41.209
C05974=1016.094,236.776,-143.061,-24.402,21.388,-41.207
C05975=1016.096,236.991,-143.086,-24.402,21.388,-41.207
C05976=1016.099,237.205,-143.110,-24.403,21.388,-41.205
C05977=1016.101,237.419,-143.135,-24.403,21.388,-41.203
C05978=1016.103,237.634,-143.160,-24.403,21.388,-41.201
C05979=1016.106,237.882,-143.189,-24.403,21.388,-41.199
C05980=1016.109,238.130,-143.217,-24.404,21.387,-41.197
C05981=1016.112,238.378,-143.246,-24.404,21.387,-41.195
C05982=1016.115,238.626,-143.275,-24.405,21.388,-41.192
C05983=1016.117,238.875,-143.304,-24.405,21.387,-41.190
C05984=1016.121,239.123,-143.333,-24.405,21.387,-41.188
C05985=1016.123,239.372,-143.361,-24.405,21.387,-41.186
C05986=1016.126,239.620,-143.390,-24.406,21.387,-41.184
C05987=1016.129,239.868,-143.419,-24.406,21.386,-41.183
C05988=1016.132,240.117,-143.447,-24.406,21.386,-41.181
C05989=1016.135,240.365,-143.476,-24.406,21.386,-41.179
C05990=1016.137,240.613,-143.506,-24.407,21.386,-41.177
C05991=1016.140,240.862,-143.534,-24.407,21.386,-41.174
C05992=1016.143,241.110,-143.563,-24.407,21.386,-41.172
C05993=1016.146,241.358,-143.592,-24.408,21.386,-41.170
C05994=1016.148,241.607,-143.621,-24.408,21.386,-41.168
C05995=1016.152,241.855,-143.649,-24.408,21.385,-41.166
C05996=1016.155,242.103,-143.678,-24.408,21.385,-41.164
C05997=1016.157,242.351,-143.707,-24.409,21.385,-41.162
C05998=1016.161,242.600,-143.736,-24.409,21.385,-41.159
C05999=1016.163,242.843,-143.765,-24.410,21.385,-41.157
C06000=1016.167,243.086,-143.793,-24.410,21.385,-41.155
C06001=1016.169,243.330,-143.821,-24.410,21.385,-41.153
C06002=1016.172,243.572,-143.849,-24.410,21.384,-41.151
C06003=1016.175,243.816,-143.878,-24.411,21.384,-41.150
C06004=1016.178,244.059,-143.906,-24.411,21.384,-41.148
C06005=1016.181,244.303,-143.934,-24.411,21.384,-41.144
C06006=1016.184,244.545,-143.963,-24.412,21.384,-41.143
C06007=1016.186,244.793,-143.992,-24.412,21.384,-41.141
C06008=1016.190,245.042,-144.021,-24.412,21.384,-41.139
C06009=1016.193,245.290,-144.051,-24.412,21.384,-41.137
C06010=1016.196,245.538,-144.079,-24.413,21.384,-41.134
C06011=1016.199,245.787,-144.109,-24.413,21.384,-41.132
C06012=1016.202,246.035,-144.138,-24.413,21.383,-41.129
C06013=1016.205,246.284,-144.167,-24.414,21.382,-41.127
C06014=1016.208,246.532,-144.195,-24.414,21.382,-41.126
C06015=1016.211,246.780,-144.224,-24.414,21.383,-41.122
C06016=1016.214,247.028,-144.253,-24.415,21.382,-41.120
C06017=1016.217,247.276,-144.282,-24.415,21.382,-41.118
C06018=1016.220,247.525,-144.312,-24.415,21.382,-41.117
C06019=1016.223,247.773,-144.341,-24.416,21.382,-41.113
C06020=1016.226,248.022,-144.370,-24.416,21.382,-41.111
C06021=1016.229,248.270,-144.399,-24.416,21.381,-41.109
C06022=1016.233,248.518,-144.429,-24.417,21.381,-41.107
C06023=1016.236,248.766,-144.458,-24.417,21.381,-41.104
C06024=1016.238,249.014,-144.488,-24.417,21.381,-41.102
C06025=1016.242,249.263,-144.517,-24.418,21.381,-41.100
C06026=1016.245,249.511,-144.546,-24.418,21.381,-41.098
C06027=1016.248,249.754,-144.574,-24.418,21.381,-41.095
C06028=1016.251,249.998,-144.603,-24.419,21.381,-41.093
C06029=1016.254,250.241,-144.631,-24.419,21.380,-41.091
C06030=1016.257,250.484,-144.660,-24.419,21.380,-41.089
C06031=1016.260,250.728,-144.690,-24.420,21.380,-41.085
C06032=1016.264,250.971,-144.718,-24.420,21.380,-41.084
C06033=1016.267,251.214,-144.747,-24.420,21.380,-41.082
C06034=1016.270,251.457,-144.775,-24.421,21.380,-41.078
C06035=1016.273,251.706,-144.805,-24.421,21.380,-41.076
C06036=1016.276,251.954,-144.834,-24.421,21.379,-41.074
C06037=1016.280,252.203,-144.864,-24.421,21.378,-41.072
C06038=1016.283,252.451,-144.892,-24.422,21.379,-41.069
C06039=1016.286,252.698,-144.923,-24.422,21.379,-41.067
C06040=1016.289,252.947,-144.952,-24.423,21.378,-41.065
C06041=1016.292,253.195,-144.981,-24.423,21.378,-41.061
C06042=1016.296,253.443,-145.011,-24.423,21.378,-41.060
C06043=1016.299,253.692,-145.040,-24.424,21.378,-41.058
C06044=1016.303,253.940,-145.069,-24.424,21.378,-41.054
C06045=1016.305,254.188,-145.100,-24.424,21.378,-41.052
C06046=1016.309,254.436,-145.128,-24.425,21.377,-41.049
C06047=1016.312,254.685,-145.158,-24.425,21.377,-41.047
C06048=1016.315,254.932,-145.188,-24.425,21.377,-41.045
C06049=1016.319,255.181,-145.217,-24.426,21.377,-41.042
C06050=1016.322,255.429,-145.246,-24.426,21.377,-41.040
C06051=1016.325,255.678,-145.277,-24.426,21.376,-41.037
C06052=1016.328,255.926,-145.305,-24.427,21.376,-41.034
C06053=1016.332,256.174,-145.336,-24.427,21.376,-41.032
C06054=1016.335,256.422,-145.365,-24.428,21.377,-41.029
C06055=1016.338,256.666,-145.394,-24.428,21.376,-41.027
C06056=1016.341,256.909,-145.423,-24.428,21.375,-41.025
C06057=1016.345,257.153,-145.452,-24.429,21.376,-41.021
C06058=1016.348,257.396,-145.481,-24.429,21.376,-41.019
C06059=1016.352,257.640,-145.510,-24.429,21.375,-41.018
C06060=1016.355,257.883,-145.539,-24.430,21.375,-41.014
C06061=1016.358,258.126,-145.569,-24.430,21.375,-41.012
C06062=1016.374,259.362,-145.722,-24.551,21.322,-40.171
C06063=1016.377,259.642,-145.759,-24.587,21.310,-39.930
C06064=1016.379,259.921,-145.796,-24.622,21.298,-39.688
C06065=1016.381,260.201,-145.833,-24.658,21.287,-39.446
C06066=1016.382,260.481,-145.871,-24.693,21.275,-39.204
C06067=1016.382,260.728,-145.906,-24.725,21.267,-38.988
C06068=1016.383,260.975,-145.941,-24.758,21.259,-38.770
C06069=1016.383,261.223,-145.977,-24.790,21.251,-38.554
C06070=1016.382,261.471,-146.013,-24.823,21.245,-38.337
C06071=1016.382,261.750,-146.054,-24.860,21.238,-38.090
C06072=1016.380,262.029,-146.095,-24.897,21.233,-37.842
C06073=1016.379,262.309,-146.138,-24.935,21.227,-37.593
C06074=1016.376,262.588,-146.182,-24.973,21.223,-37.345
C06075=1016.374,262.835,-146.220,-25.006,21.220,-37.124
C06076=1016.371,263.082,-146.260,-25.040,21.217,-36.903
C06077=1016.368,263.329,-146.301,-25.074,21.216,-36.681
C06078=1016.365,263.575,-146.341,-25.108,21.215,-36.458
C06079=1016.360,263.854,-146.386,-25.147,21.216,-36.205
C06080=1016.355,264.134,-146.434,-25.186,21.217,-35.952
C06081=1016.351,264.412,-146.482,-25.226,21.219,-35.699
C06082=1016.345,264.692,-146.529,-25.265,21.221,-35.444
C06083=1016.340,264.938,-146.573,-25.300,21.225,-35.219
C06084=1016.334,265.183,-146.616,-25.335,21.229,-34.991
C06085=1016.327,265.430,-146.660,-25.370,21.233,-34.766
C06086=1016.321,265.676,-146.705,-25.406,21.239,-34.538
C06087=1016.314,265.955,-146.756,-25.446,21.246,-34.279
C06088=1016.306,266.234,-146.809,-25.487,21.254,-34.021
C06089=1016.297,266.513,-146.861,-25.527,21.264,-33.760
C06090=1016.287,266.791,-146.915,-25.568,21.275,-33.499
C06091=1016.278,267.037,-146.962,-25.604,21.284,-33.268
C06092=1016.271,267.282,-147.011,-25.641,21.295,-33.037
C06093=1016.262,267.528,-147.059,-25.677,21.306,-32.805
C06094=1016.251,267.773,-147.108,-25.714,21.319,-32.571
C06095=1016.240,268.051,-147.165,-25.755,21.334,-32.305
C06096=1016.229,268.330,-147.222,-25.797,21.350,-32.039
C06097=1016.216,268.608,-147.280,-25.839,21.367,-31.772
C06098=1016.203,268.886,-147.338,-25.881,21.386,-31.502
C06099=1016.191,269.131,-147.390,-25.918,21.402,-31.266
C06100=1016.180,269.375,-147.443,-25.955,21.420,-31.029
C06101=1016.168,269.619,-147.495,-25.992,21.438,-30.791
C06102=1016.155,269.863,-147.549,-26.030,21.459,-30.551
C06103=1016.140,270.142,-147.611,-26.072,21.483,-30.277
C06104=1016.125,270.420,-147.673,-26.115,21.507,-30.003
C06105=1016.109,270.698,-147.736,-26.158,21.533,-29.728
C06106=1016.093,270.976,-147.800,-26.201,21.560,-29.450
C06107=1016.078,271.220,-147.856,-26.238,21.585,-29.208
C06108=1016.063,271.462,-147.913,-26.276,21.610,-28.964
C06109=1016.048,271.705,-147.970,-26.314,21.637,-28.720
C06110=1016.032,271.948,-148.028,-26.351,21.664,-28.476
C06111=1016.014,272.226,-148.095,-26.395,21.697,-28.194
C06112=1015.993,272.504,-148.163,-26.438,21.731,-27.910
C06113=1015.975,272.782,-148.231,-26.481,21.766,-27.626
C06114=1015.955,273.060,-148.300,-26.525,21.803,-27.342
C06115=1015.937,273.302,-148.361,-26.562,21.835,-27.092
C06116=1015.919,273.543,-148.423,-26.600,21.869,-26.841
C06117=1015.900,273.786,-148.484,-26.638,21.904,-26.589
C06118=1015.881,274.027,-148.546,-26.676,21.940,-26.336
C06119=1015.859,274.305,-148.618,-26.720,21.983,-26.043
C06120=1015.836,274.583,-148.692,-26.763,22.026,-25.749
C06121=1015.813,274.860,-148.766,-26.807,22.073,-25.453
C06122=1015.789,275.138,-148.839,-26.851,22.119,-25.156
C06123=1015.768,275.378,-148.906,-26.889,22.162,-24.896
C06124=1015.747,275.618,-148.970,-26.927,22.204,-24.635
C06125=1015.725,275.859,-149.037,-26.965,22.250,-24.373
C06126=1015.702,276.099,-149.104,-27.003,22.295,-24.109
C06127=1015.676,276.376,-149.182,-27.046,22.349,-23.804
C06128=1015.650,276.654,-149.260,-27.090,22.404,-23.496
C06129=1015.623,276.930,-149.340,-27.134,22.462,-23.186
C06130=1015.596,277.207,-149.420,-27.177,22.521,-22.877
C06131=1015.571,277.446,-149.490,-27.215,22.573,-22.606
C06132=1015.546,277.684,-149.559,-27.252,22.626,-22.334
C06133=1015.521,277.923,-149.630,-27.290,22.681,-22.062
C06134=1015.496,278.162,-149.702,-27.327,22.737,-21.789
C06135=1015.466,278.439,-149.786,-27.370,22.804,-21.469
C06136=1015.435,278.715,-149.869,-27.413,22.872,-21.148
C06137=1015.404,278.991,-149.955,-27.456,22.942,-20.824
C06138=1015.372,279.268,-150.040,-27.498,23.014,-20.499
C06139=1015.344,279.505,-150.115,-27.534,23.078,-20.218
C06140=1015.316,279.742,-150.190,-27.570,23.143,-19.936
C06141=1015.288,279.978,-150.265,-27.606,23.208,-19.653
C06142=1015.259,280.215,-150.341,-27.642,23.276,-19.367
C06143=1015.225,280.492,-150.430,-27.684,23.357,-19.031
C06144=1015.190,280.768,-150.521,-27.725,23.440,-18.691
C06145=1015.155,281.043,-150.612,-27.766,23.526,-18.349
C06146=1015.118,281.319,-150.703,-27.807,23.613,-18.004
C06147=1015.088,281.554,-150.782,-27.842,23.690,-17.706
C06148=1015.056,281.790,-150.862,-27.877,23.768,-17.406
C06149=1015.025,282.023,-150.942,-27.911,23.848,-17.104
C06150=1014.993,282.259,-151.023,-27.945,23.929,-16.801
C06151=1014.954,282.534,-151.118,-27.984,24.027,-16.441
C06152=1014.915,282.809,-151.214,-28.023,24.128,-16.079
C06153=1014.876,283.084,-151.312,-28.062,24.232,-15.713
C06154=1014.835,283.359,-151.409,-28.100,24.338,-15.343
C06155=1014.800,283.592,-151.493,-28.132,24.429,-15.026
C06156=1014.765,283.824,-151.577,-28.164,24.524,-14.708
C06157=1014.730,284.057,-151.663,-28.195,24.619,-14.388
C06158=1014.694,284.289,-151.748,-28.226,24.716,-14.065
C06159=1014.651,284.563,-151.850,-28.261,24.835,-13.680
C06160=1014.607,284.837,-151.952,-28.296,24.955,-13.292
C06161=1014.563,285.111,-152.057,-28.330,25.079,-12.901
C06162=1014.519,285.385,-152.160,-28.364,25.204,-12.507
C06163=1014.480,285.615,-152.249,-28.391,25.314,-12.171
C06164=1014.442,285.845,-152.339,-28.418,25.425,-11.832
C06165=1014.403,286.076,-152.429,-28.444,25.537,-11.492
C06166=1014.364,286.305,-152.519,-28.470,25.652,-11.148
C06167=1014.316,286.578,-152.628,-28.499,25.792,-10.737
C06168=1014.267,286.851,-152.737,-28.527,25.935,-10.321
C06169=1014.218,287.123,-152.847,-28.555,26.082,-9.899
C06170=1014.169,287.395,-152.959,-28.581,26.233,-9.471
C06171=1014.127,287.623,-153.052,-28.602,26.363,-9.109
C06172=1014.084,287.850,-153.147,-28.622,26.495,-8.743
C06173=1014.041,288.077,-153.242,-28.641,26.630,-8.372
C06174=1013.997,288.305,-153.338,-28.659,26.767,-7.999
C06175=1013.945,288.577,-153.453,-28.679,26.937,-7.545
C06176=1013.891,288.847,-153.569,-28.698,27.109,-7.088
C06177=1013.838,289.118,-153.687,-28.715,27.285,-6.624
C06178=1013.783,289.388,-153.805,-28.730,27.467,-6.153
C06179=1013.738,289.613,-153.904,-28.742,27.622,-5.757
C06180=1013.691,289.837,-154.004,-28.752,27.779,-5.357
C06181=1013.644,290.061,-154.105,-28.760,27.939,-4.952
C06182=1013.597,290.286,-154.206,-28.767,28.103,-4.544
C06183=1013.538,290.554,-154.328,-28.773,28.305,-4.046
C06184=1013.480,290.823,-154.452,-28.777,28.512,-3.541
C06185=1013.420,291.091,-154.578,-28.778,28.722,-3.030
C06186=1013.361,291.359,-154.703,-28.777,28.937,-2.514
C06187=1013.310,291.581,-154.808,-28.773,29.120,-2.080
C06188=1013.260,291.802,-154.914,-28.768,29.306,-1.642
C06189=1013.208,292.023,-155.020,-28.760,29.494,-1.200
C06190=1013.157,292.242,-155.127,-28.751,29.686,-0.753
C06191=1013.093,292.510,-155.258,-28.736,29.926,-0.203
C06192=1013.029,292.775,-155.390,-28.717,30.168,0.353
C06193=1012.964,293.041,-155.522,-28.695,30.417,0.916
C06194=1012.898,293.307,-155.656,-28.669,30.673,1.490
C06195=1012.843,293.524,-155.767,-28.645,30.886,1.967
C06196=1012.789,293.742,-155.878,-28.617,31.104,2.450
C06197=1012.733,293.958,-155.990,-28.586,31.327,2.940
C06198=1012.677,294.175,-156.103,-28.552,31.552,3.436
C06199=1012.608,294.438,-156.243,-28.506,31.835,4.050
C06200=1012.537,294.701,-156.382,-28.455,32.123,4.674
C06201=1012.467,294.964,-156.524,-28.398,32.417,5.306
C06202=1012.394,295.226,-156.666,-28.335,32.716,5.947
C06203=1012.336,295.439,-156.783,-28.280,32.966,6.479
C06204=1012.276,295.652,-156.900,-28.220,33.220,7.016
C06205=1012.216,295.864,-157.018,-28.156,33.478,7.560
C06206=1012.155,296.075,-157.138,-28.087,33.740,8.111
C06207=1012.079,296.335,-157.286,-27.996,34.068,8.799
C06208=1012.003,296.595,-157.435,-27.897,34.404,9.500
C06209=1011.925,296.855,-157.585,-27.790,34.746,10.213
C06210=1011.847,297.113,-157.736,-27.675,35.094,10.935
C06211=1011.783,297.321,-157.859,-27.576,35.380,11.529
C06212=1011.719,297.529,-157.983,-27.470,35.670,12.129
C06213=1011.653,297.736,-158.107,-27.359,35.965,12.738
C06214=1011.587,297.943,-158.233,-27.241,36.263,13.354
C06215=1011.505,298.199,-158.391,-27.085,36.641,14.134
C06216=1011.422,298.454,-158.549,-26.918,37.024,14.926
C06217=1011.338,298.709,-158.708,-26.741,37.414,15.733
C06218=1011.252,298.963,-158.869,-26.551,37.810,16.553
C06219=1011.183,299.166,-158.999,-26.391,38.132,17.220
C06220=1011.114,299.368,-159.129,-26.221,38.458,17.898
C06221=1011.044,299.569,-159.260,-26.044,38.787,18.584
C06222=1010.973,299.769,-159.392,-25.858,39.121,19.281
///RCONF 0,0,0,0,0,0,0,0,0,0,0,0,0,0,0,0,0,0,0,0,0,0,0,0
C06223=1010.884,300.021,-159.559,-25.611,39.544,20.170
C06224=1010.793,300.272,-159.727,-25.349,39.974,21.077
C06225=1010.702,300.522,-159.896,-25.071,40.409,21.999
C06226=1010.609,300.770,-160.068,-24.778,40.847,22.938
C06227=1010.535,300.967,-160.203,-24.533,41.199,23.695
C06228=1010.460,301.163,-160.340,-24.278,41.553,24.463
C06229=1010.386,301.358,-160.478,-24.010,41.911,25.245
C06230=1010.310,301.553,-160.617,-23.731,42.271,26.037
C06231=1010.213,301.798,-160.793,-23.359,42.732,27.060
C06232=1010.115,302.044,-160.972,-22.967,43.196,28.105
C06233=1010.016,302.287,-161.152,-22.552,43.665,29.173
C06234=1009.916,302.530,-161.332,-22.115,44.137,30.264
C06235=1009.837,302.720,-161.475,-21.757,44.508,31.133
C06236=1009.757,302.909,-161.618,-21.384,44.880,32.017
C06237=1009.677,303.097,-161.763,-20.996,45.254,32.916
C06238=1009.596,303.284,-161.908,-20.592,45.628,33.828
C06239=1009.491,303.525,-162.095,-20.052,46.107,35.019
C06240=1009.386,303.762,-162.283,-19.485,46.587,36.235
C06241=1009.279,304.000,-162.473,-18.890,47.066,37.479
C06242=1009.171,304.237,-162.664,-18.265,47.545,38.750
C06243=1009.087,304.419,-162.814,-17.761,47.914,39.754
C06244=1009.002,304.600,-162.964,-17.237,48.283,40.777
C06245=1008.917,304.781,-163.115,-16.695,48.650,41.816
C06246=1008.831,304.961,-163.266,-16.132,49.015,42.875
C06247=1008.717,305.193,-163.464,-15.372,49.485,44.275
C06248=1008.604,305.425,-163.663,-14.578,49.950,45.708
C06249=1008.490,305.654,-163.863,-13.751,50.408,47.169
C06250=1008.374,305.884,-164.065,-12.888,50.859,48.662
C06251=1008.285,306.058,-164.219,-12.202,51.199,49.829
C06252=1008.195,306.231,-164.375,-11.496,51.534,51.012
C06253=1008.104,306.404,-164.532,-10.767,51.863,52.216
C06254=1008.013,306.576,-164.690,-10.017,52.187,53.438
C06255=1007.893,306.800,-164.898,-9.002,52.599,55.068
C06256=1007.772,307.024,-165.107,-7.948,53.000,56.733
C06257=1007.649,307.245,-165.317,-6.854,53.388,58.434
C06258=1007.526,307.464,-165.530,-5.724,53.761,60.165
C06259=1007.432,307.631,-165.691,-4.837,54.035,61.506
C06260=1007.337,307.796,-165.852,-3.930,54.299,62.863
C06261=1007.241,307.960,-166.016,-2.999,54.554,64.242
C06262=1007.145,308.124,-166.180,-2.047,54.798,65.640
C06263=1007.017,308.339,-166.397,-0.758,55.103,67.512
C06264=1006.889,308.552,-166.615,0.564,55.388,69.411
C06265=1006.759,308.765,-166.835,1.921,55.651,71.337
C06266=1006.628,308.975,-167.056,3.305,55.891,73.285
C06267=1006.537,309.119,-167.209,4.272,56.043,74.635
C06268=1006.447,309.262,-167.362,5.252,56.184,75.995
C06269=1006.354,309.404,-167.514,6.248,56.313,77.368
C06270=1006.253,309.544,-167.662,7.250,56.430,78.743
C06271=1006.586,309.681,-168.032,8.024,56.512,79.800
C06272=1006.713,309.515,-167.860,6.823,56.382,78.159
C06273=1006.828,309.346,-167.680,5.634,56.235,76.523
C06274=1006.937,309.177,-167.499,4.460,56.071,74.897
C06275=1007.045,309.006,-167.316,3.305,55.891,73.285
C06276=1007.175,308.795,-167.095,1.921,55.651,71.337
C06277=1007.305,308.582,-166.875,0.564,55.388,69.411
C06278=1007.434,308.369,-166.656,-0.758,55.103,67.512
C06279=1007.562,308.154,-166.439,-2.047,54.798,65.640
C06280=1007.658,307.990,-166.275,-2.999,54.554,64.242
C06281=1007.753,307.827,-166.113,-3.930,54.299,62.863
C06282=1007.848,307.661,-165.950,-4.837,54.035,61.506
C06283=1007.942,307.494,-165.789,-5.724,53.761,60.165
C06284=1008.066,307.275,-165.577,-6.854,53.388,58.434
C06285=1008.188,307.054,-165.367,-7.948,53.000,56.733
C06286=1008.310,306.830,-165.158,-9.002,52.599,55.068
C06287=1008.430,306.606,-164.950,-10.018,52.186,53.439
C06288=1008.521,306.434,-164.792,-10.767,51.863,52.216
C06289=1008.611,306.261,-164.635,-11.496,51.534,51.012
C06290=1008.701,306.087,-164.479,-12.202,51.199,49.829
C06291=1008.791,305.914,-164.324,-12.888,50.859,48.662
C06292=1008.906,305.684,-164.122,-13.751,50.408,47.169
C06293=1009.021,305.455,-163.922,-14.580,49.949,45.706
C06294=1009.134,305.224,-163.723,-15.374,49.484,44.273
C06295=1009.247,304.991,-163.525,-16.133,49.014,42.872
C06296=1009.333,304.811,-163.374,-16.695,48.650,41.816
C06297=1009.418,304.630,-163.223,-17.238,48.282,40.774
C06298=1009.503,304.449,-163.073,-17.761,47.914,39.754
C06299=1009.588,304.267,-162.924,-18.265,47.545,38.750
C06300=1009.695,304.031,-162.732,-18.890,47.066,37.479
C06301=1009.801,303.793,-162.543,-19.485,46.587,36.235
C06302=1009.908,303.555,-162.355,-20.052,46.107,35.019
C06303=1010.012,303.315,-162.167,-20.592,45.628,33.828
C06304=1010.093,303.127,-162.022,-20.996,45.254,32.916
C06305=1010.173,302.939,-161.878,-21.384,44.880,32.017
C06306=1010.253,302.751,-161.734,-21.757,44.508,31.133
C06307=1010.333,302.560,-161.592,-22.115,44.137,30.264
C06308=1010.432,302.318,-161.410,-22.552,43.665,29.173
C06309=1010.531,302.074,-161.231,-22.967,43.196,28.105
C06310=1010.629,301.828,-161.053,-23.359,42.732,27.060
C06311=1010.726,301.583,-160.877,-23.731,42.271,26.037
C06312=1010.802,301.388,-160.738,-24.011,41.910,25.243
C06313=1010.877,301.193,-160.600,-24.278,41.553,24.463
C06314=1010.951,300.997,-160.463,-24.533,41.199,23.695
C06315=1011.025,300.801,-160.327,-24.778,40.847,22.938
C06316=1011.118,300.552,-160.156,-25.071,40.409,21.999
C06317=1011.209,300.302,-159.986,-25.349,39.974,21.077
C06318=1011.300,300.052,-159.818,-25.611,39.544,20.170
///RCONF 0,0,0,0,1,0,0,0,0,0,0,0,0,0,0,0,0,0,0,0,0,0,0,0
C06319=1011.389,299.800,-159.651,-25.858,39.121,19.281
C06320=1011.460,299.599,-159.520,-26.044,38.787,18.584
C06321=1011.529,299.397,-159.389,-26.221,38.458,17.898
C06322=1011.599,299.195,-159.258,-26.391,38.132,17.220
C06323=1011.668,298.993,-159.128,-26.551,37.810,16.553
C06324=1011.753,298.739,-158.967,-26.741,37.414,15.733
C06325=1011.838,298.484,-158.807,-26.918,37.024,14.926
C06326=1011.921,298.229,-158.650,-27.085,36.640,14.133
C06327=1012.003,297.972,-158.493,-27.241,36.263,13.354
C06328=1012.070,297.766,-158.367,-27.359,35.964,12.737
C06329=1012.134,297.558,-158.243,-27.470,35.670,12.129
C06330=1012.198,297.351,-158.118,-27.576,35.380,11.529
C06331=1012.262,297.143,-157.995,-27.675,35.094,10.935
C06332=1012.341,296.885,-157.844,-27.790,34.746,10.213
C06333=1012.418,296.626,-157.694,-27.897,34.404,9.500
C06334=1012.495,296.366,-157.545,-27.996,34.068,8.799
C06335=1012.571,296.106,-157.397,-28.087,33.740,8.111
C06336=1012.631,295.894,-157.278,-28.156,33.478,7.560
C06337=1012.691,295.682,-157.159,-28.220,33.220,7.016
C06338=1012.751,295.470,-157.042,-28.280,32.966,6.479
C06339=1012.811,295.257,-156.925,-28.335,32.716,5.947
C06340=1012.882,294.994,-156.783,-28.398,32.417,5.306
C06341=1012.954,294.731,-156.642,-28.455,32.123,4.674
C06342=1013.023,294.468,-156.501,-28.506,31.835,4.050
C06343=1013.093,294.204,-156.363,-28.552,31.552,3.436
C06344=1013.149,293.988,-156.250,-28.586,31.327,2.940
C06345=1013.204,293.771,-156.138,-28.617,31.104,2.450
C06346=1013.260,293.555,-156.026,-28.645,30.886,1.967
C06347=1013.314,293.337,-155.915,-28.669,30.673,1.490
C06348=1013.379,293.071,-155.781,-28.695,30.417,0.916
C06349=1013.445,292.806,-155.649,-28.717,30.168,0.353
C06350=1013.509,292.540,-155.516,-28.736,29.926,-0.203
C06351=1013.572,292.273,-155.386,-28.751,29.686,-0.753
C06352=1013.624,292.053,-155.279,-28.760,29.494,-1.200
C06353=1013.676,291.832,-155.173,-28.768,29.306,-1.642
C06354=1013.727,291.611,-155.068,-28.773,29.120,-2.080
C06355=1013.776,291.389,-154.962,-28.777,28.937,-2.514
C06356=1013.836,291.122,-154.836,-28.778,28.722,-3.030
C06357=1013.895,290.853,-154.712,-28.777,28.511,-3.540
C06358=1013.954,290.585,-154.588,-28.773,28.305,-4.046
C06359=1014.012,290.315,-154.466,-28.767,28.103,-4.544
C06360=1014.059,290.092,-154.364,-28.760,27.939,-4.952
C06361=1014.106,289.867,-154.263,-28.752,27.779,-5.357
C06362=1014.152,289.643,-154.164,-28.742,27.622,-5.757
C06363=1014.199,289.418,-154.063,-28.730,27.467,-6.153
C06364=1014.254,289.148,-153.945,-28.715,27.285,-6.624
C06365=1014.308,288.878,-153.828,-28.698,27.109,-7.088
C06366=1014.360,288.606,-153.711,-28.679,26.937,-7.545
C06367=1014.413,288.335,-153.596,-28.659,26.767,-7.999
C06368=1014.457,288.107,-153.501,-28.641,26.630,-8.372
C06369=1014.499,287.880,-153.406,-28.622,26.495,-8.743
C06370=1014.542,287.653,-153.311,-28.602,26.363,-9.109
C06371=1014.584,287.425,-153.218,-28.581,26.233,-9.471
C06372=1014.634,287.153,-153.106,-28.555,26.082,-9.899
C06373=1014.682,286.881,-152.996,-28.527,25.935,-10.321
C06374=1014.731,286.608,-152.887,-28.499,25.792,-10.737
C06375=1014.778,286.336,-152.778,-28.470,25.652,-11.148
C06376=1014.818,286.105,-152.687,-28.444,25.537,-11.492
C06377=1014.857,285.875,-152.598,-28.418,25.425,-11.832
C06378=1014.895,285.645,-152.508,-28.391,25.314,-12.171
C06379=1014.934,285.415,-152.420,-28.364,25.204,-12.507
C06380=1014.979,285.141,-152.315,-28.330,25.079,-12.901
C06381=1015.022,284.867,-152.212,-28.296,24.955,-13.292
C06382=1015.066,284.593,-152.109,-28.261,24.835,-13.680
C06383=1015.109,284.319,-152.007,-28.226,24.716,-14.065
C06384=1015.145,284.087,-151.921,-28.195,24.619,-14.388
C06385=1015.180,283.854,-151.836,-28.164,24.524,-14.708
C06386=1015.214,283.621,-151.752,-28.132,24.429,-15.026
C06387=1015.250,283.389,-151.668,-28.100,24.338,-15.343
C06388=1015.290,283.113,-151.570,-28.062,24.232,-15.713
C06389=1015.330,282.839,-151.473,-28.023,24.128,-16.079
C06390=1015.369,282.564,-151.377,-27.984,24.027,-16.441
C06391=1015.407,282.288,-151.281,-27.945,23.929,-16.801
C06392=1015.439,282.054,-151.200,-27.911,23.848,-17.104
C06393=1015.471,281.820,-151.121,-27.877,23.768,-17.406
C06394=1015.502,281.585,-151.041,-27.842,23.690,-17.706
C06395=1015.533,281.349,-150.962,-27.807,23.613,-18.004
C06396=1015.569,281.074,-150.870,-27.766,23.526,-18.349
C06397=1015.605,280.798,-150.779,-27.725,23.440,-18.691
C06398=1015.639,280.522,-150.689,-27.684,23.357,-19.031
C06399=1015.674,280.246,-150.599,-27.642,23.276,-19.367
C06400=1015.703,280.009,-150.523,-27.606,23.208,-19.653
C06401=1015.731,279.772,-150.448,-27.570,23.143,-19.936
C06402=1015.759,279.535,-150.373,-27.534,23.078,-20.218
C06403=1015.787,279.298,-150.299,-27.498,23.014,-20.499
C06404=1015.818,279.022,-150.213,-27.456,22.942,-20.824
C06405=1015.850,278.745,-150.129,-27.413,22.872,-21.148
C06406=1015.880,278.469,-150.044,-27.370,22.804,-21.469
C06407=1015.910,278.192,-149.960,-27.327,22.737,-21.789
C06408=1015.935,277.953,-149.889,-27.290,22.681,-22.062
C06409=1015.961,277.715,-149.818,-27.252,22.626,-22.334
C06410=1015.985,277.476,-149.748,-27.215,22.573,-22.606
C06411=1016.009,277.237,-149.678,-27.177,22.521,-22.877
C06412=1016.037,276.961,-149.598,-27.134,22.462,-23.186
C06413=1016.064,276.683,-149.519,-27.090,22.404,-23.496
C06414=1016.091,276.406,-149.441,-27.046,22.349,-23.804
C06415=1016.116,276.128,-149.362,-27.003,22.294,-24.111
C06416=1016.139,275.888,-149.296,-26.965,22.250,-24.373
C06417=1016.161,275.648,-149.229,-26.927,22.204,-24.635
C06418=1016.183,275.408,-149.163,-26.889,22.162,-24.896
C06419=1016.203,275.167,-149.098,-26.851,22.119,-25.156
C06420=1016.227,274.890,-149.024,-26.807,22.073,-25.453
C06421=1016.250,274.613,-148.950,-26.763,22.026,-25.749
C06422=1016.273,274.335,-148.876,-26.720,21.983,-26.043
C06423=1016.295,274.057,-148.805,-26.676,21.940,-26.336
C06424=1016.314,273.815,-148.743,-26.638,21.904,-26.589
C06425=1016.333,273.573,-148.681,-26.600,21.869,-26.841
C06426=1016.351,273.332,-148.619,-26.562,21.835,-27.092
C06427=1016.369,273.090,-148.558,-26.525,21.803,-27.342
C06428=1016.389,272.812,-148.489,-26.481,21.766,-27.626
C06429=1016.407,272.534,-148.421,-26.438,21.731,-27.910
C06430=1016.428,272.256,-148.353,-26.395,21.697,-28.194
C06431=1016.446,271.978,-148.286,-26.351,21.664,-28.476
C06432=1016.462,271.735,-148.228,-26.314,21.637,-28.720
C06433=1016.477,271.492,-148.171,-26.276,21.610,-28.964
C06434=1016.492,271.250,-148.114,-26.238,21.585,-29.208
C06435=1016.507,271.006,-148.058,-26.201,21.560,-29.450
C06436=1016.522,270.728,-147.994,-26.158,21.533,-29.728
C06437=1016.538,270.450,-147.931,-26.115,21.507,-30.003
C06438=1016.554,270.172,-147.869,-26.072,21.483,-30.277
C06439=1016.569,269.893,-147.807,-26.030,21.459,-30.551
C06440=1016.581,269.649,-147.754,-25.992,21.438,-30.791
C06441=1016.593,269.405,-147.701,-25.955,21.420,-31.029
C06442=1016.605,269.161,-147.648,-25.918,21.402,-31.266
C06443=1016.617,268.916,-147.596,-25.881,21.386,-31.502
C06444=1016.630,268.638,-147.538,-25.839,21.367,-31.772
C06445=1016.642,268.359,-147.479,-25.797,21.350,-32.039
C06446=1016.653,268.080,-147.423,-25.755,21.333,-32.307
C06447=1016.665,267.802,-147.366,-25.713,21.318,-32.573
C06448=1016.674,267.556,-147.317,-25.677,21.306,-32.805
C06449=1016.684,267.312,-147.268,-25.641,21.295,-33.037
C06450=1016.692,267.067,-147.220,-25.604,21.284,-33.269
C06451=1016.700,266.821,-147.172,-25.568,21.275,-33.499
C06452=1016.710,266.542,-147.119,-25.527,21.264,-33.760
C06453=1016.718,266.264,-147.067,-25.487,21.254,-34.021
C06454=1016.726,265.985,-147.015,-25.446,21.246,-34.279
C06455=1016.734,265.706,-146.962,-25.406,21.239,-34.538
C06456=1016.741,265.460,-146.918,-25.370,21.233,-34.766
C06457=1016.746,265.215,-146.874,-25.335,21.229,-34.991
C06458=1016.752,264.968,-146.830,-25.300,21.225,-35.219
C06459=1016.758,264.721,-146.787,-25.265,21.221,-35.444
C06460=1016.764,264.442,-146.739,-25.226,21.219,-35.699
C06461=1016.768,264.164,-146.691,-25.186,21.217,-35.952
C06462=1016.773,263.885,-146.644,-25.147,21.216,-36.205
C06463=1016.777,263.605,-146.598,-25.108,21.215,-36.458
C06464=1016.781,263.359,-146.558,-25.074,21.216,-36.681
C06465=1016.784,263.112,-146.517,-25.040,21.217,-36.903
C06466=1016.786,262.865,-146.477,-25.006,21.220,-37.124
C06467=1016.789,262.618,-146.439,-24.973,21.223,-37.345
C06468=1016.790,262.339,-146.396,-24.935,21.227,-37.593
C06469=1016.792,262.060,-146.353,-24.897,21.233,-37.842
C06470=1016.793,261.780,-146.311,-24.860,21.238,-38.090
C06471=1016.795,261.501,-146.269,-24.823,21.245,-38.337
C06472=1016.795,261.253,-146.233,-24.790,21.251,-38.554
C06473=1016.796,261.006,-146.198,-24.758,21.259,-38.770
C06474=1016.795,260.758,-146.163,-24.725,21.267,-38.988
C06475=1016.794,260.510,-146.128,-24.693,21.275,-39.204
C06476=1016.793,260.231,-146.090,-24.658,21.287,-39.446
C06477=1016.791,259.951,-146.052,-24.622,21.298,-39.688
C06478=1016.789,259.672,-146.016,-24.587,21.310,-39.930
C06479=1016.787,259.392,-145.979,-24.551,21.322,-40.171
C06480=1016.770,258.156,-145.825,-24.430,21.375,-41.012
C06481=1016.766,257.913,-145.796,-24.430,21.375,-41.014
C06482=1016.763,257.669,-145.767,-24.429,21.375,-41.018
C06483=1016.760,257.426,-145.738,-24.429,21.376,-41.019
C06484=1016.757,257.182,-145.709,-24.429,21.376,-41.021
C06485=1016.753,256.939,-145.680,-24.428,21.375,-41.025
C06486=1016.750,256.695,-145.651,-24.428,21.376,-41.027
C06487=1016.747,256.452,-145.622,-24.428,21.377,-41.029
C06488=1016.743,256.204,-145.592,-24.427,21.376,-41.032
C06489=1016.740,255.955,-145.562,-24.427,21.376,-41.034
C06490=1016.737,255.708,-145.533,-24.426,21.376,-41.037
C06491=1016.733,255.459,-145.503,-24.426,21.377,-41.040
C06492=1016.730,255.211,-145.474,-24.426,21.377,-41.042
C06493=1016.727,254.963,-145.444,-24.425,21.377,-41.045
C06494=1016.723,254.715,-145.415,-24.425,21.377,-41.047
C06495=1016.720,254.466,-145.385,-24.425,21.377,-41.049
C06496=1016.717,254.218,-145.356,-24.424,21.378,-41.052
C06497=1016.714,253.969,-145.326,-24.424,21.378,-41.054
C06498=1016.710,253.722,-145.297,-24.424,21.378,-41.058
C06499=1016.707,253.473,-145.267,-24.423,21.378,-41.060
C06500=1016.703,253.226,-145.237,-24.423,21.378,-41.061
C06501=1016.700,252.977,-145.208,-24.423,21.378,-41.065
C06502=1016.697,252.729,-145.179,-24.422,21.379,-41.067
C06503=1016.694,252.480,-145.149,-24.422,21.379,-41.069
C06504=1016.690,252.232,-145.120,-24.421,21.378,-41.072
C06505=1016.688,251.984,-145.090,-24.421,21.379,-41.074
C06506=1016.684,251.735,-145.061,-24.421,21.380,-41.076
C06507=1016.681,251.487,-145.032,-24.421,21.380,-41.078
C06508=1016.678,251.244,-145.003,-24.420,21.380,-41.082
C06509=1016.675,251.001,-144.974,-24.420,21.380,-41.084
C06510=1016.671,250.757,-144.946,-24.420,21.380,-41.085
C06511=1016.668,250.514,-144.916,-24.419,21.380,-41.089
C06512=1016.665,250.271,-144.888,-24.419,21.380,-41.091
C06513=1016.662,250.028,-144.859,-24.419,21.381,-41.093
C06514=1016.659,249.784,-144.831,-24.418,21.381,-41.095
C06515=1016.655,249.541,-144.802,-24.418,21.381,-41.098
C06516=1016.653,249.292,-144.773,-24.418,21.381,-41.100
C06517=1016.650,249.044,-144.744,-24.417,21.381,-41.102
C06518=1016.647,248.795,-144.714,-24.417,21.381,-41.104
C06519=1016.643,248.548,-144.685,-24.417,21.381,-41.107
C06520=1016.640,248.300,-144.655,-24.416,21.381,-41.109
C06521=1016.637,248.051,-144.626,-24.416,21.382,-41.111
C06522=1016.634,247.803,-144.597,-24.416,21.382,-41.113
C06523=1016.631,247.555,-144.568,-24.415,21.382,-41.117
C06524=1016.628,247.307,-144.539,-24.415,21.382,-41.118
C06525=1016.624,247.058,-144.510,-24.415,21.382,-41.120
C06526=1016.621,246.810,-144.481,-24.414,21.383,-41.122
C06527=1016.619,246.562,-144.451,-24.414,21.382,-41.126
C06528=1016.615,246.314,-144.423,-24.414,21.382,-41.127
C06529=1016.613,246.065,-144.393,-24.413,21.383,-41.129
C06530=1016.609,245.817,-144.364,-24.413,21.384,-41.132
C06531=1016.606,245.569,-144.335,-24.413,21.384,-41.134
C06532=1016.603,245.320,-144.307,-24.412,21.384,-41.137
C06533=1016.601,245.072,-144.277,-24.412,21.384,-41.139
C06534=1016.597,244.823,-144.248,-24.412,21.384,-41.141
C06535=1016.594,244.575,-144.219,-24.412,21.384,-41.143
C06536=1016.591,244.332,-144.190,-24.411,21.384,-41.144
C06537=1016.588,244.089,-144.163,-24.411,21.384,-41.148
C06538=1016.586,243.846,-144.134,-24.411,21.384,-41.150
C06539=1016.582,243.603,-144.105,-24.410,21.384,-41.151
C06540=1016.580,243.359,-144.077,-24.410,21.385,-41.153
C06541=1016.577,243.116,-144.048,-24.410,21.385,-41.155
C06542=1016.574,242.873,-144.021,-24.410,21.385,-41.157
C06543=1016.571,242.629,-143.992,-24.409,21.385,-41.159
C06544=1016.568,242.381,-143.963,-24.409,21.385,-41.162
C06545=1016.565,242.133,-143.934,-24.408,21.385,-41.164
C06546=1016.562,241.884,-143.905,-24.408,21.385,-41.166
C06547=1016.559,241.636,-143.877,-24.408,21.386,-41.168
C06548=1016.557,241.388,-143.847,-24.408,21.386,-41.170
C06549=1016.554,241.140,-143.819,-24.407,21.386,-41.172
C06550=1016.551,240.891,-143.790,-24.407,21.386,-41.174
C06551=1016.548,240.643,-143.761,-24.407,21.386,-41.177
C06552=1016.545,240.395,-143.732,-24.406,21.386,-41.179
C06553=1016.542,240.146,-143.704,-24.406,21.386,-41.181
C06554=1016.539,239.899,-143.675,-24.406,21.386,-41.183
C06555=1016.537,239.650,-143.645,-24.406,21.387,-41.184
C06556=1016.534,239.402,-143.617,-24.405,21.387,-41.186
C06557=1016.530,239.154,-143.589,-24.405,21.387,-41.188
C06558=1016.528,238.905,-143.559,-24.405,21.387,-41.190
C06559=1016.525,238.657,-143.531,-24.405,21.388,-41.192
C06560=1016.522,238.409,-143.502,-24.404,21.387,-41.195
C06561=1016.519,238.160,-143.474,-24.404,21.387,-41.197
C06562=1016.517,237.912,-143.444,-24.403,21.388,-41.199
C06563=1016.514,237.663,-143.416,-24.403,21.388,-41.201
C06564=1016.509,237.306,-143.375,-24.403,21.388,-41.203
C06565=1016.506,236.948,-143.334,-24.402,21.388,-41.207
C06566=1016.501,236.591,-143.292,-24.402,21.389,-41.209
C06567=1016.498,236.233,-143.251,-24.402,21.389,-41.212
C06568=1016.495,235.985,-143.222,-24.401,21.389,-41.214
C06569=1016.492,235.736,-143.193,-24.401,21.389,-41.216
C06570=1016.490,235.489,-143.165,-24.401,21.389,-41.218
C06571=1016.487,235.240,-143.137,-24.401,21.389,-41.219
C06572=1016.484,234.992,-143.108,-24.400,21.389,-41.221
C06573=1016.481,234.744,-143.079,-24.400,21.390,-41.223
C06574=1016.479,234.495,-143.050,-24.400,21.390,-41.225
C06575=1016.476,234.247,-143.022,-24.400,21.390,-41.227
C06576=1016.473,233.998,-142.994,-24.399,21.390,-41.229
C06577=1016.470,233.750,-142.965,-24.399,21.390,-41.231
C06578=1016.468,233.502,-142.937,-24.399,21.391,-41.233
C06579=1016.466,233.253,-142.908,-24.399,21.391,-41.234
C06580=1016.462,233.005,-142.879,-24.398,21.390,-41.236
C06581=1016.459,232.756,-142.851,-24.398,21.390,-41.238
C06582=1016.457,232.508,-142.823,-24.398,21.391,-41.240
C06583=1016.455,232.260,-142.794,-24.397,21.391,-41.242
C06584=1016.451,231.883,-142.751,-24.397,21.390,-41.245
C06585=1016.446,231.505,-142.707,-24.397,21.392,-41.247
C06586=1016.443,231.128,-142.665,-24.396,21.391,-41.251
C06587=1016.438,230.752,-142.621,-24.396,21.391,-41.252
C06588=1016.437,230.509,-142.594,-24.396,21.392,-41.254
C06589=1016.434,230.266,-142.566,-24.395,21.392,-41.256
C06590=1016.432,230.023,-142.538,-24.395,21.392,-41.258
C06591=1016.429,229.779,-142.511,-24.395,21.392,-41.260
C06592=1016.426,229.537,-142.483,-24.395,21.392,-41.262
C06593=1016.424,229.294,-142.455,-24.394,21.392,-41.263
C06594=1016.421,229.051,-142.427,-24.394,21.392,-41.265
C06595=1016.419,228.808,-142.400,-24.394,21.393,-41.266
C06596=1016.417,228.559,-142.371,-24.394,21.393,-41.267
C06597=1016.414,228.311,-142.343,-24.394,21.393,-41.269
C06598=1016.412,228.063,-142.315,-24.393,21.394,-41.271
C06599=1016.409,227.815,-142.286,-24.393,21.393,-41.273
C06600=1016.406,227.566,-142.258,-24.393,21.393,-41.275
C06601=1016.404,227.318,-142.230,-24.393,21.393,-41.276
C06602=1016.401,227.069,-142.202,-24.392,21.394,-41.278
C06603=1016.398,226.821,-142.174,-24.392,21.394,-41.280
C06604=1016.397,226.572,-142.145,-24.392,21.393,-41.282
C06605=1016.394,226.324,-142.117,-24.391,21.393,-41.284
C06606=1016.391,226.075,-142.089,-24.391,21.394,-41.285
C06607=1016.389,225.827,-142.061,-24.391,21.395,-41.286
C06608=1016.386,225.578,-142.033,-24.391,21.395,-41.288
C06609=1016.384,225.330,-142.005,-24.391,21.394,-41.289
C06610=1016.382,225.082,-141.977,-24.390,21.394,-41.291
C06611=1016.380,224.833,-141.948,-24.390,21.395,-41.293
C06612=1016.377,224.585,-141.920,-24.390,21.395,-41.295
C06613=1016.374,224.336,-141.892,-24.390,21.395,-41.297
C06614=1016.372,224.088,-141.864,-24.389,21.394,-41.298
C06615=1016.369,223.840,-141.835,-24.389,21.395,-41.300
C06616=1016.367,223.597,-141.809,-24.389,21.395,-41.300
C06617=1016.365,223.354,-141.781,-24.389,21.396,-41.302
C06618=1016.362,223.111,-141.753,-24.389,21.396,-41.304
C06619=1016.360,222.868,-141.726,-24.388,21.395,-41.306
C06620=1016.358,222.626,-141.698,-24.388,21.395,-41.308
C06621=1016.356,222.383,-141.671,-24.388,21.396,-41.309
C06622=1016.353,222.140,-141.644,-24.388,21.397,-41.310
C06623=1016.352,221.897,-141.616,-24.388,21.396,-41.311
C06624=1016.349,221.649,-141.588,-24.387,21.396,-41.313
C06625=1016.346,221.400,-141.560,-24.387,21.396,-41.315
C06626=1016.345,221.152,-141.532,-24.387,21.397,-41.317
C06627=1016.342,220.904,-141.504,-24.386,21.396,-41.318
C06628=1016.340,220.655,-141.477,-24.386,21.396,-41.320
C06629=1016.337,220.406,-141.448,-24.386,21.397,-41.321
C06630=1016.335,220.158,-141.420,-24.386,21.397,-41.323
C06631=1016.333,219.910,-141.392,-24.386,21.397,-41.324
C06632=1016.330,219.662,-141.364,-24.385,21.397,-41.326
C06633=1016.328,219.414,-141.336,-24.385,21.397,-41.328
C06634=1016.326,219.164,-141.308,-24.385,21.397,-41.330
C06635=1016.324,218.916,-141.281,-24.385,21.397,-41.330
C06636=1016.322,218.667,-141.252,-24.385,21.397,-41.332
C06637=1016.319,218.420,-141.224,-24.384,21.398,-41.333
C06638=1016.317,218.171,-141.197,-24.384,21.398,-41.335
C06639=1016.315,217.922,-141.169,-24.384,21.397,-41.337
C06640=1016.313,217.674,-141.141,-24.384,21.397,-41.339
C06641=1016.310,217.425,-141.112,-24.384,21.398,-41.339
C06642=1016.308,217.177,-141.085,-24.383,21.399,-41.341
C06643=1016.306,216.929,-141.058,-24.383,21.398,-41.342
C06644=1016.304,216.686,-141.030,-24.383,21.398,-41.344
C06645=1016.302,216.444,-141.003,-24.383,21.398,-41.346
C06646=1016.300,216.200,-140.976,-24.383,21.398,-41.346
C06647=1016.298,215.958,-140.949,-24.382,21.399,-41.348
C06648=1016.296,215.715,-140.921,-24.382,21.399,-41.350
C06649=1016.294,215.473,-140.894,-24.382,21.399,-41.352
C06650=1016.292,215.229,-140.867,-24.382,21.398,-41.353
C06651=1016.289,214.987,-140.840,-24.382,21.399,-41.354
C06652=1016.287,214.738,-140.812,-24.381,21.400,-41.356
C06653=1016.285,214.489,-140.785,-24.381,21.399,-41.357
C06654=1016.283,214.242,-140.757,-24.381,21.399,-41.359
C06655=1016.281,213.993,-140.729,-24.381,21.400,-41.359
C06656=1016.278,213.744,-140.701,-24.381,21.400,-41.361
C06657=1016.277,213.496,-140.673,-24.380,21.400,-41.363
C06658=1016.275,213.247,-140.646,-24.380,21.400,-41.365
C06659=1016.272,213.000,-140.618,-24.380,21.400,-41.366
C06660=1016.270,212.750,-140.590,-24.380,21.400,-41.366
C06661=1016.268,212.502,-140.563,-24.380,21.400,-41.368
C06662=1016.267,212.253,-140.535,-24.379,21.400,-41.370
C06663=1016.264,212.005,-140.507,-24.379,21.400,-41.372
C06664=1016.262,211.757,-140.480,-24.379,21.401,-41.372
C06665=1016.260,211.508,-140.452,-24.379,21.401,-41.374
C06666=1016.258,211.260,-140.425,-24.378,21.400,-41.375
C06667=1016.256,211.011,-140.396,-24.378,21.400,-41.377
C06668=1016.254,210.763,-140.369,-24.378,21.401,-41.378
C06669=1016.252,210.515,-140.342,-24.378,21.401,-41.379
C06670=1016.250,210.265,-140.314,-24.378,21.401,-41.381
C06671=1016.248,210.018,-140.286,-24.377,21.401,-41.383
C06672=1016.246,209.775,-140.260,-24.377,21.401,-41.383
C06673=1016.244,209.533,-140.233,-24.377,21.401,-41.385
C06674=1016.242,209.290,-140.205,-24.377,21.402,-41.387
C06675=1016.240,209.047,-140.179,-24.377,21.401,-41.388
C06676=1016.238,208.805,-140.152,-24.377,21.402,-41.389
C06677=1016.236,208.562,-140.125,-24.376,21.402,-41.391
C06678=1016.234,208.319,-140.098,-24.376,21.401,-41.392
C06679=1016.233,208.076,-140.071,-24.376,21.402,-41.392
C06680=1016.230,207.828,-140.043,-24.376,21.402,-41.394
C06681=1016.228,207.579,-140.016,-24.376,21.402,-41.396
C06682=1016.227,207.330,-139.989,-24.375,21.402,-41.398
C06683=1016.225,207.083,-139.961,-24.375,21.402,-41.398
C06684=1016.223,206.834,-139.933,-24.375,21.402,-41.399
C06685=1016.221,206.585,-139.906,-24.375,21.402,-41.401
C06686=1016.219,206.337,-139.879,-24.375,21.402,-41.401
C06687=1016.218,206.089,-139.851,-24.375,21.403,-41.403
C06688=1016.215,205.840,-139.824,-24.374,21.403,-41.405
C06689=1016.214,205.592,-139.796,-24.374,21.402,-41.407
C06690=1016.212,205.343,-139.769,-24.374,21.403,-41.407
C06691=1016.210,205.095,-139.742,-24.374,21.403,-41.409
C06692=1016.208,204.846,-139.714,-24.373,21.403,-41.410
C06693=1016.206,204.598,-139.687,-24.374,21.404,-41.411
C06694=1016.205,204.349,-139.659,-24.373,21.403,-41.412
C06695=1016.203,204.101,-139.632,-24.373,21.403,-41.414
C06696=1016.201,203.852,-139.605,-24.373,21.404,-41.415
C06697=1016.199,203.604,-139.577,-24.373,21.403,-41.416
C06698=1016.193,202.387,-139.442,-24.425,21.378,-41.051
C06699=1016.192,202.000,-139.398,-24.424,21.378,-41.052
C06700=1016.193,201.652,-139.360,-24.424,21.378,-41.054
C06701=1016.193,201.300,-139.321,-24.424,21.378,-41.058
C06702=1016.194,200.893,-139.277,-24.423,21.379,-41.060
C06703=1016.194,200.665,-139.252,-24.423,21.378,-41.061
C06704=1016.194,200.436,-139.227,-24.423,21.378,-41.063
C06705=1016.195,200.213,-139.202,-24.423,21.378,-41.065
C06706=1016.195,200.001,-139.179,-24.423,21.378,-41.065
C06707=1016.197,199.600,-139.136,-24.422,21.379,-41.069
C06708=1016.197,199.210,-139.093,-24.422,21.379,-41.071
C06709=1016.198,198.812,-139.049,-24.421,21.379,-41.074
C06710=1016.198,198.411,-139.005,-24.421,21.379,-41.076
C06711=1016.199,198.010,-138.962,-24.421,21.380,-41.078
C06712=1016.200,197.609,-138.917,-24.420,21.380,-41.082
C06713=1016.201,197.208,-138.874,-24.420,21.380,-41.084
C06714=1016.202,196.807,-138.831,-24.419,21.380,-41.087
C06715=1016.202,196.406,-138.787,-24.419,21.380,-41.089
C06716=1016.204,196.005,-138.743,-24.419,21.381,-41.091
C06717=1016.204,195.604,-138.699,-24.418,21.380,-41.094
C06718=1016.205,195.203,-138.655,-24.418,21.381,-41.097
C06719=1016.206,194.802,-138.612,-24.418,21.381,-41.100
C06720=1016.206,194.401,-138.569,-24.417,21.381,-41.102
C06721=1016.208,193.999,-138.525,-24.417,21.381,-41.105
C06722=1016.209,193.598,-138.481,-24.417,21.382,-41.108
C06723=1016.209,193.197,-138.437,-24.416,21.382,-41.109
C06724=1016.210,192.796,-138.394,-24.416,21.382,-41.113
C06725=1016.210,192.395,-138.351,-24.415,21.382,-41.115
C06726=1016.212,191.993,-138.307,-24.415,21.382,-41.118
C06727=1016.213,191.592,-138.264,-24.415,21.382,-41.120
C06728=1016.213,191.191,-138.220,-24.414,21.382,-41.124
C06729=1016.215,190.790,-138.177,-24.414,21.383,-41.126
C06730=1016.215,190.390,-138.133,-24.414,21.383,-41.128
C06731=1016.216,189.988,-138.090,-24.413,21.383,-41.131
C06732=1016.217,189.587,-138.046,-24.413,21.383,-41.133
C06733=1016.219,189.186,-138.003,-24.412,21.384,-41.137
C06734=1016.220,188.785,-137.960,-24.412,21.384,-41.139
C06735=1016.220,188.384,-137.916,-24.412,21.384,-41.141
C06736=1016.221,187.983,-137.873,-24.411,21.384,-41.144
C06737=1016.222,187.582,-137.830,-24.411,21.385,-41.146
C06738=1016.223,187.181,-137.787,-24.411,21.384,-41.150
C06739=1016.224,186.780,-137.744,-24.410,21.384,-41.151
C06740=1016.225,186.379,-137.701,-24.410,21.384,-41.155
C06741=1016.226,185.978,-137.657,-24.410,21.385,-41.157
C06742=1016.228,185.577,-137.615,-24.409,21.385,-41.159
C06743=1016.229,185.175,-137.571,-24.409,21.385,-41.162
C06744=1016.231,184.775,-137.528,-24.409,21.386,-41.165
C06745=1016.231,184.374,-137.485,-24.408,21.386,-41.168
C06746=1016.232,183.973,-137.442,-24.408,21.386,-41.170
C06747=1016.233,183.572,-137.399,-24.407,21.386,-41.172
C06748=1016.235,183.172,-137.356,-24.407,21.386,-41.176
C06749=1016.236,182.770,-137.313,-24.407,21.387,-41.177
C06750=1016.237,182.369,-137.270,-24.406,21.386,-41.181
C06751=1016.238,181.968,-137.227,-24.406,21.387,-41.183
C06752=1016.239,181.567,-137.184,-24.405,21.387,-41.186
C06753=1016.239,181.167,-137.141,-24.405,21.387,-41.188
C06754=1016.241,180.766,-137.098,-24.405,21.387,-41.190
C06755=1016.242,180.365,-137.056,-24.404,21.388,-41.194
C06756=1016.243,179.964,-137.013,-24.404,21.388,-41.196
C06757=1016.244,179.563,-136.970,-24.403,21.388,-41.199
C06758=1016.246,179.163,-136.927,-24.403,21.388,-41.201
C06759=1016.247,178.762,-136.885,-24.403,21.388,-41.205
C06760=1016.248,178.360,-136.841,-24.402,21.388,-41.207
C06761=1016.249,177.960,-136.798,-24.402,21.389,-41.209
C06762=1016.251,177.559,-136.756,-24.402,21.389,-41.212
C06763=1016.252,177.158,-136.713,-24.401,21.389,-41.214
C06764=1016.253,176.758,-136.671,-24.401,21.389,-41.218
C06765=1016.255,176.357,-136.628,-24.401,21.389,-41.219
C06766=1016.255,175.956,-136.585,-24.400,21.390,-41.223
C06767=1016.257,175.555,-136.542,-24.400,21.390,-41.225
C06768=1016.258,175.154,-136.500,-24.400,21.390,-41.227
C06769=1016.259,174.754,-136.458,-24.399,21.390,-41.231
C06770=1016.260,174.353,-136.415,-24.399,21.391,-41.233
C06771=1016.262,173.952,-136.372,-24.398,21.390,-41.236
C06772=1016.263,173.552,-136.329,-24.398,21.390,-41.238
C06773=1016.264,173.152,-136.287,-24.397,21.391,-41.242
C06774=1016.266,172.750,-136.245,-24.397,21.391,-41.243
C06775=1016.267,172.350,-136.202,-24.397,21.391,-41.247
C06776=1016.269,171.949,-136.160,-24.396,21.392,-41.249
C06777=1016.270,171.549,-136.118,-24.396,21.392,-41.251
C06778=1016.272,171.148,-136.076,-24.396,21.392,-41.254
C06779=1016.273,170.748,-136.033,-24.395,21.392,-41.256
C06780=1016.273,170.347,-135.990,-24.395,21.392,-41.260
C06781=1016.275,169.946,-135.948,-24.395,21.392,-41.262
C06782=1016.277,169.547,-135.905,-24.394,21.392,-41.265
C06783=1016.278,169.146,-135.864,-24.394,21.393,-41.267
C06784=1016.279,168.745,-135.821,-24.393,21.393,-41.271
C06785=1016.280,168.344,-135.779,-24.393,21.393,-41.273
C06786=1016.282,167.945,-135.737,-24.393,21.394,-41.275
C06787=1016.284,167.543,-135.694,-24.392,21.394,-41.278
C06788=1016.284,167.143,-135.652,-24.392,21.394,-41.280
C06789=1016.287,166.743,-135.610,-24.391,21.393,-41.284
C06790=1016.287,166.343,-135.568,-24.391,21.395,-41.286
C06791=1016.290,165.942,-135.526,-24.391,21.394,-41.289
C06792=1016.290,165.542,-135.484,-24.390,21.394,-41.291
C06793=1016.292,165.141,-135.441,-24.390,21.395,-41.295
C06794=1016.293,164.741,-135.399,-24.390,21.395,-41.297
C06795=1016.295,164.341,-135.357,-24.389,21.395,-41.300
C06796=1016.296,163.955,-135.316,-24.389,21.395,-41.302
C06797=1016.297,163.766,-135.297,-24.389,21.395,-41.304
C06798=1016.298,163.353,-135.253,-24.388,21.396,-41.306
C06799=1016.299,163.117,-135.229,-24.388,21.395,-41.308
C06800=1016.299,162.864,-135.202,-24.388,21.396,-41.309
C06801=1016.301,162.601,-135.175,-24.388,21.396,-41.311
C06802=1016.302,162.332,-135.147,-24.387,21.396,-41.313
C06803=1016.303,162.061,-135.118,-24.387,21.396,-41.315
C06804=1016.304,161.791,-135.089,-24.387,21.397,-41.317
C06805=1016.304,161.529,-135.062,-24.387,21.397,-41.319
C06806=1016.305,161.278,-135.036,-24.386,21.396,-41.320
C06807=1016.307,161.041,-135.012,-24.386,21.396,-41.322
C06808=1016.308,160.816,-134.988,-24.386,21.397,-41.324
C06809=1016.308,160.603,-134.965,-24.386,21.397,-41.325
C06810=1016.309,160.197,-134.923,-24.385,21.397,-41.328
C06811=1016.311,159.801,-134.881,-24.385,21.397,-41.330
C06812=1016.317,159.401,-134.843,-24.384,21.398,-41.333
C06813=1016.324,159.000,-134.803,-24.384,21.398,-41.335
C06814=1016.330,158.599,-134.765,-24.384,21.397,-41.339
C06815=1016.337,158.197,-134.727,-24.383,21.399,-41.341
C06816=1016.345,157.794,-134.688,-24.383,21.398,-41.344
C06817=1016.351,157.391,-134.649,-24.383,21.398,-41.346
C06818=1016.358,156.987,-134.610,-24.382,21.399,-41.350
C06819=1016.365,156.582,-134.572,-24.382,21.399,-41.352
C06820=1016.372,156.176,-134.532,-24.381,21.399,-41.355
C06821=1016.377,155.899,-134.506,-24.381,21.399,-41.357
C06822=1016.381,155.622,-134.479,-24.381,21.399,-41.359
C06823=1016.386,155.362,-134.454,-24.381,21.399,-41.361
C06824=1016.393,154.953,-134.415,-24.380,21.400,-41.363
C06825=1016.399,154.544,-134.376,-24.380,21.400,-41.366
C06826=1016.406,154.134,-134.336,-24.380,21.400,-41.368
C06827=1016.413,153.724,-134.297,-24.379,21.401,-41.372
C06828=1016.421,153.312,-134.258,-24.378,21.400,-41.375
C06829=1016.427,152.900,-134.218,-24.378,21.400,-41.377
C06830=1016.434,152.488,-134.179,-24.378,21.401,-41.381
C06831=1016.440,152.076,-134.139,-24.377,21.401,-41.383
C06832=1016.447,151.663,-134.099,-24.377,21.402,-41.387
C06833=1016.454,151.249,-134.059,-24.377,21.402,-41.389
C06834=1016.460,150.836,-134.020,-24.376,21.401,-41.392
C06835=1016.467,150.422,-133.981,-24.376,21.402,-41.394
C06836=1016.474,150.008,-133.940,-24.375,21.402,-41.398
C06837=1016.481,149.594,-133.901,-24.375,21.402,-41.401
C06838=1016.488,149.180,-133.861,-24.375,21.403,-41.403
C06839=1016.494,148.766,-133.821,-24.374,21.403,-41.407
C06840=1016.501,148.352,-133.782,-24.374,21.403,-41.409
C06841=1016.508,147.938,-133.742,-24.373,21.403,-41.412
C06842=1016.514,147.524,-133.703,-24.373,21.403,-41.416
C06843=1016.521,147.111,-133.663,-24.372,21.404,-41.418
C06844=1016.527,146.697,-133.623,-24.372,21.404,-41.422
C06845=1016.534,146.284,-133.584,-24.372,21.404,-41.424
C06846=1016.541,145.871,-133.544,-24.371,21.405,-41.427
C06847=1016.547,145.459,-133.505,-24.371,21.404,-41.431
C06848=1016.553,145.047,-133.466,-24.370,21.405,-41.432
C06849=1016.560,144.634,-133.426,-24.370,21.405,-41.436
C06850=1016.566,144.224,-133.386,-24.370,21.405,-41.438
C06851=1016.573,143.814,-133.347,-24.369,21.406,-41.442
C06852=1016.579,143.405,-133.308,-24.369,21.405,-41.445
C06853=1016.585,142.996,-133.269,-24.368,21.406,-41.448
C06854=1016.591,142.587,-133.230,-24.368,21.406,-41.451
C06855=1016.597,142.181,-133.191,-24.368,21.406,-41.453
C06856=1016.603,141.774,-133.152,-24.367,21.407,-41.457
C06857=1016.611,141.369,-133.114,-24.366,21.406,-41.460
C06858=1016.616,140.965,-133.075,-24.366,21.407,-41.462
C06859=1016.622,140.547,-133.035,-24.366,21.408,-41.466
C06860=1016.626,140.311,-133.012,-24.366,21.408,-41.468
C06861=1016.630,140.053,-132.987,-24.365,21.408,-41.470
C06862=1016.634,139.776,-132.961,-24.365,21.408,-41.471
C06863=1016.639,139.488,-132.933,-24.365,21.408,-41.473
C06864=1016.642,139.200,-132.906,-24.364,21.408,-41.475
C06865=1016.648,138.923,-132.879,-24.364,21.407,-41.476
C06866=1016.651,138.663,-132.855,-24.364,21.408,-41.478
C06867=1016.654,138.426,-132.832,-24.364,21.408,-41.480
C06868=1016.658,138.209,-132.811,-24.363,21.408,-41.482
C06869=1016.661,138.003,-132.791,-24.363,21.408,-41.484
C06870=1016.666,137.602,-132.753,-24.363,21.408,-41.486
C06871=1016.672,137.232,-132.718,-24.363,21.410,-41.488
C06872=1016.677,136.896,-132.686,-24.362,21.409,-41.491
C06873=1016.682,136.579,-132.655,-24.361,21.409,-41.495
C06874=1016.686,136.262,-132.625,-24.361,21.410,-41.497
C06875=1016.691,135.922,-132.593,-24.361,21.409,-41.500
C06876=1016.697,135.550,-132.557,-24.360,21.410,-41.502
C06877=1016.702,135.155,-132.519,-24.360,21.411,-41.505
C06878=1016.708,134.757,-132.481,-24.360,21.410,-41.508
C06879=1016.714,134.358,-132.443,-24.359,21.411,-41.510
C06880=1016.720,133.959,-132.405,-24.359,21.411,-41.514
C06881=1016.725,133.561,-132.367,-24.358,21.411,-41.517
C06882=1016.731,133.162,-132.329,-24.358,21.412,-41.519
C06883=1016.737,132.763,-132.291,-24.358,21.411,-41.523
C06884=1016.743,132.364,-132.253,-24.357,21.412,-41.525
C06885=1016.748,131.966,-132.215,-24.357,21.412,-41.528
C06886=1016.754,131.567,-132.177,-24.356,21.412,-41.532
C06887=1016.759,131.168,-132.140,-24.356,21.413,-41.534
C06888=1016.765,130.770,-132.101,-24.356,21.413,-41.538
C06889=1016.771,130.371,-132.063,-24.355,21.413,-41.541
C06890=1016.777,129.973,-132.026,-24.355,21.413,-41.543
C06891=1016.782,129.574,-131.987,-24.354,21.413,-41.547
C06892=1016.787,129.176,-131.950,-24.354,21.413,-41.550
C06893=1016.793,128.777,-131.912,-24.354,21.414,-41.552
C06894=1016.798,128.378,-131.873,-24.353,21.414,-41.555
C06895=1016.804,127.980,-131.835,-24.353,21.415,-41.558
C06896=1016.810,127.581,-131.798,-24.352,21.414,-41.561
C06897=1016.815,127.182,-131.759,-24.352,21.415,-41.565
C06898=1016.820,126.784,-131.722,-24.351,21.415,-41.567
C06899=1016.825,126.386,-131.684,-24.351,21.415,-41.571
C06900=1016.831,125.987,-131.646,-24.350,21.415,-41.574
C06901=1016.836,125.588,-131.608,-24.350,21.416,-41.576
C06902=1016.842,125.190,-131.570,-24.350,21.416,-41.580
C06903=1016.847,124.791,-131.532,-24.349,21.416,-41.583
C06904=1016.852,124.393,-131.494,-24.349,21.416,-41.585
C06905=1016.857,123.994,-131.456,-24.348,21.417,-41.589
C06906=1016.863,123.595,-131.418,-24.348,21.416,-41.592
C06907=1016.868,123.197,-131.380,-24.348,21.418,-41.595
C06908=1016.873,122.798,-131.343,-24.347,21.417,-41.598
C06909=1016.879,122.400,-131.306,-24.347,21.418,-41.602
C06910=1016.884,122.002,-131.268,-24.346,21.417,-41.605
C06911=1016.889,121.603,-131.229,-24.346,21.418,-41.607
C06912=1016.894,121.205,-131.191,-24.345,21.418,-41.611
C06913=1016.899,120.806,-131.154,-24.345,21.418,-41.614
C06914=1016.904,120.408,-131.116,-24.345,21.419,-41.617
C06915=1016.910,120.009,-131.078,-24.344,21.419,-41.620
C06916=1016.916,119.611,-131.040,-24.343,21.419,-41.624
C06917=1016.921,119.212,-131.003,-24.343,21.420,-41.626
C06918=1016.927,118.814,-130.966,-24.343,21.420,-41.629
C06919=1016.932,118.415,-130.928,-24.342,21.420,-41.633
C06920=1016.937,118.016,-130.891,-24.342,21.420,-41.637
C06921=1016.943,117.618,-130.854,-24.341,21.420,-41.638
C06922=1016.948,117.220,-130.816,-24.341,21.421,-41.642
C06923=1016.954,116.821,-130.778,-24.340,21.420,-41.646
C06924=1016.959,116.423,-130.740,-24.340,21.421,-41.649
C06925=1016.965,116.024,-130.703,-24.340,21.422,-41.652
C06926=1016.970,115.625,-130.665,-24.339,21.422,-41.655
C06927=1016.975,115.227,-130.628,-24.339,21.422,-41.659
C06928=1016.980,114.828,-130.591,-24.338,21.422,-41.662
C06929=1016.986,114.431,-130.553,-24.338,21.423,-41.664
C06930=1016.991,114.032,-130.516,-24.337,21.422,-41.668
C06931=1016.996,113.633,-130.478,-24.337,21.423,-41.671
C06932=1017.001,113.235,-130.441,-24.336,21.423,-41.675
C06933=1017.007,112.836,-130.403,-24.336,21.423,-41.677
C06934=1017.012,112.438,-130.366,-24.335,21.424,-41.681
C06935=1017.017,112.039,-130.328,-24.335,21.423,-41.684
C06936=1017.022,111.641,-130.292,-24.334,21.424,-41.688
C06937=1017.027,111.243,-130.254,-24.334,21.425,-41.690
C06938=1017.032,110.844,-130.216,-24.334,21.425,-41.694
C06939=1017.037,110.445,-130.179,-24.333,21.425,-41.697
C06940=1017.043,110.047,-130.141,-24.333,21.425,-41.701
C06941=1017.047,109.648,-130.104,-24.332,21.426,-41.703
C06942=1017.053,109.249,-130.066,-24.332,21.426,-41.707
C06943=1017.057,108.851,-130.030,-24.331,21.426,-41.710
C06944=1017.062,108.452,-129.992,-24.331,21.426,-41.714
C06945=1017.068,108.054,-129.955,-24.330,21.426,-41.717
C06946=1017.073,107.654,-129.917,-24.330,21.427,-41.719
C06947=1017.077,107.257,-129.880,-24.330,21.427,-41.723
C06948=1017.082,106.858,-129.842,-24.329,21.427,-41.727
C06949=1017.087,106.459,-129.805,-24.328,21.427,-41.730
C06950=1017.092,106.061,-129.768,-24.328,21.428,-41.734
C06951=1017.097,105.662,-129.730,-24.328,21.428,-41.736
C06952=1017.102,105.264,-129.693,-24.327,21.429,-41.740
C06953=1017.106,104.865,-129.656,-24.327,21.429,-41.743
C06954=1017.112,104.466,-129.619,-24.326,21.429,-41.747
C06955=1017.117,104.067,-129.581,-24.326,21.429,-41.751
C06956=1017.121,103.669,-129.544,-24.325,21.430,-41.754
C06957=1017.126,103.270,-129.507,-24.325,21.430,-41.756
C06958=1017.131,102.872,-129.470,-24.324,21.430,-41.760
C06959=1017.136,102.473,-129.432,-24.324,21.430,-41.763
C06960=1017.140,102.074,-129.395,-24.323,21.430,-41.767
C06961=1017.145,101.676,-129.358,-24.323,21.431,-41.771
C06962=1017.150,101.276,-129.320,-24.322,21.431,-41.775
C06963=1017.154,100.878,-129.283,-24.322,21.431,-41.778
C06964=1017.160,100.479,-129.246,-24.322,21.432,-41.780
C06965=1017.164,100.080,-129.209,-24.321,21.432,-41.784
C06966=1017.168,99.681,-129.171,-24.320,21.432,-41.787
C06967=1017.173,99.283,-129.135,-24.320,21.432,-41.791
C06968=1017.178,98.884,-129.097,-24.319,21.433,-41.795
C06969=1017.182,98.485,-129.060,-24.319,21.432,-41.798
C06970=1017.186,98.086,-129.023,-24.318,21.433,-41.802
C06971=1017.192,97.688,-128.986,-24.318,21.433,-41.806
C06972=1017.196,97.288,-128.949,-24.318,21.434,-41.808
C06973=1017.201,96.889,-128.912,-24.317,21.434,-41.811
C06974=1017.205,96.490,-128.874,-24.317,21.435,-41.815
C06975=1017.209,96.092,-128.837,-24.316,21.435,-41.819
C06976=1017.214,95.693,-128.800,-24.316,21.435,-41.822
C06977=1017.219,95.294,-128.763,-24.315,21.435,-41.826
C06978=1017.223,94.896,-128.726,-24.315,21.436,-41.830
C06979=1017.228,94.496,-128.689,-24.314,21.435,-41.833
C06980=1017.232,94.097,-128.652,-24.313,21.436,-41.837
C06981=1017.236,93.698,-128.615,-24.313,21.436,-41.841
C06982=1017.241,93.299,-128.577,-24.312,21.437,-41.844
C06983=1017.245,92.900,-128.540,-24.312,21.437,-41.846
C06984=1017.249,92.501,-128.504,-24.312,21.437,-41.850
C06985=1017.253,92.102,-128.467,-24.311,21.438,-41.854
C06986=1017.258,91.703,-128.429,-24.311,21.438,-41.857
C06987=1017.262,91.304,-128.392,-24.310,21.438,-41.861
C06988=1017.267,90.904,-128.356,-24.310,21.438,-41.865
C06989=1017.270,90.505,-128.318,-24.309,21.439,-41.868
C06990=1017.274,90.106,-128.281,-24.309,21.439,-41.872
C06991=1017.279,89.708,-128.245,-24.308,21.439,-41.875
C06992=1017.283,89.315,-128.208,-24.308,21.439,-41.879
C06993=1017.287,88.928,-128.172,-24.307,21.440,-41.883
C06994=1017.291,88.545,-128.137,-24.307,21.440,-41.887
C06995=1017.295,88.163,-128.101,-24.306,21.440,-41.890
C06996=1017.299,87.774,-128.065,-24.305,21.440,-41.894
C06997=1017.303,87.378,-128.029,-24.305,21.441,-41.898
C06998=1017.308,86.975,-127.991,-24.304,21.441,-41.901
C06999=1017.312,86.569,-127.954,-24.304,21.442,-41.905
C07000=1017.316,86.162,-127.917,-24.303,21.441,-41.908
C07001=1017.320,85.753,-127.878,-24.303,21.442,-41.912
C07002=1017.324,85.342,-127.840,-24.302,21.442,-41.916
C07003=1017.328,84.930,-127.802,-24.302,21.443,-41.920
C07004=1017.333,84.515,-127.764,-24.301,21.443,-41.923
C07005=1017.337,84.100,-127.726,-24.301,21.443,-41.927
C07006=1017.341,83.683,-127.687,-24.300,21.444,-41.931
C07007=1017.345,83.263,-127.649,-24.300,21.444,-41.935
C07008=1017.349,82.843,-127.610,-24.299,21.444,-41.938
C07009=1017.352,82.633,-127.590,-24.299,21.444,-41.940
C07010=1017.354,82.422,-127.571,-24.299,21.444,-41.942
C07011=1017.355,82.210,-127.551,-24.299,21.445,-41.944
C07012=1017.358,81.999,-127.532,-24.298,21.444,-41.947
C07013=1017.359,81.787,-127.512,-24.298,21.445,-41.949
C07014=1017.362,81.576,-127.493,-24.298,21.445,-41.951
C07015=1017.364,81.364,-127.473,-24.297,21.445,-41.953
C07016=1017.365,81.151,-127.454,-24.297,21.445,-41.955
C07017=1017.368,80.938,-127.434,-24.297,21.445,-41.956
C07018=1017.370,80.725,-127.415,-24.297,21.446,-41.958
C07019=1017.372,80.512,-127.395,-24.296,21.446,-41.960
C07020=1017.374,80.300,-127.375,-24.296,21.446,-41.962
C07021=1017.376,80.088,-127.355,-24.296,21.446,-41.964
C07022=1017.378,79.878,-127.337,-24.296,21.447,-41.966
C07023=1017.382,79.463,-127.298,-24.295,21.447,-41.970
C07024=1017.386,79.058,-127.261,-24.294,21.447,-41.973
C07025=1017.390,78.661,-127.224,-24.294,21.447,-41.977
C07026=1017.393,78.270,-127.189,-24.293,21.448,-41.980
C07027=1017.397,77.883,-127.153,-24.293,21.447,-41.986
C07028=1017.401,77.498,-127.117,-24.292,21.448,-41.989
C07029=1017.404,77.109,-127.082,-24.292,21.449,-41.994
C07030=1017.408,76.714,-127.045,-24.291,21.449,-41.997
C07031=1017.412,76.312,-127.008,-24.291,21.449,-42.001
C07032=1017.415,75.901,-126.970,-24.290,21.450,-42.004
C07033=1017.419,75.481,-126.933,-24.290,21.450,-42.008
C07034=1017.421,75.268,-126.913,-24.289,21.451,-42.010
C07035=1017.423,75.055,-126.893,-24.289,21.451,-42.012
C07036=1017.425,74.841,-126.874,-24.289,21.450,-42.015
C07037=1017.427,74.628,-126.854,-24.288,21.451,-42.017
C07038=1017.429,74.415,-126.835,-24.288,21.451,-42.019
C07039=1017.430,74.202,-126.815,-24.288,21.451,-42.021
C07040=1017.432,73.990,-126.795,-24.288,21.451,-42.023
C07041=1017.435,73.778,-126.776,-24.287,21.452,-42.025
C07042=1017.438,73.359,-126.738,-24.287,21.452,-42.028
C07043=1017.442,72.941,-126.699,-24.286,21.452,-42.034
C07044=1017.445,72.525,-126.662,-24.285,21.452,-42.037
C07045=1017.449,72.111,-126.623,-24.285,21.453,-42.041
C07046=1017.453,71.699,-126.586,-24.285,21.453,-42.045
C07047=1017.456,71.288,-126.548,-24.284,21.454,-42.049
C07048=1017.460,70.877,-126.510,-24.283,21.453,-42.054
C07049=1017.463,70.467,-126.473,-24.283,21.454,-42.058
C07050=1017.467,70.055,-126.436,-24.282,21.454,-42.061
C07051=1017.471,69.644,-126.398,-24.282,21.455,-42.065
C07052=1017.474,69.233,-126.361,-24.281,21.455,-42.069
C07053=1017.477,68.825,-126.323,-24.280,21.455,-42.074
C07054=1017.481,68.417,-126.287,-24.280,21.456,-42.078
C07055=1017.484,68.012,-126.249,-24.279,21.456,-42.082
C07056=1017.487,67.607,-126.212,-24.279,21.457,-42.085
C07057=1017.491,67.204,-126.175,-24.278,21.457,-42.089
C07058=1017.494,66.801,-126.139,-24.278,21.457,-42.094
C07059=1017.498,66.400,-126.102,-24.277,21.457,-42.098
C07060=1017.501,66.003,-126.067,-24.277,21.458,-42.102
C07061=1017.504,65.595,-126.029,-24.276,21.458,-42.106
C07062=1017.506,65.382,-126.009,-24.276,21.459,-42.108
C07063=1017.507,65.160,-125.989,-24.275,21.458,-42.111
C07064=1017.509,64.931,-125.969,-24.275,21.458,-42.113
C07065=1017.511,64.694,-125.947,-24.275,21.459,-42.115
C07066=1017.514,64.459,-125.926,-24.274,21.459,-42.116
C07067=1017.515,64.229,-125.905,-24.274,21.459,-42.120
C07068=1017.517,64.011,-125.886,-24.274,21.460,-42.122
C07069=1017.519,63.805,-125.866,-24.274,21.460,-42.124
C07070=1017.520,63.587,-125.847,-24.273,21.459,-42.127
C07071=1017.522,63.338,-125.824,-24.273,21.460,-42.129
C07072=1017.524,63.070,-125.800,-24.272,21.460,-42.131
C07073=1017.526,62.817,-125.777,-24.272,21.460,-42.133
C07074=1017.529,62.396,-125.739,-24.271,21.461,-42.139
C07075=1017.532,61.996,-125.703,-24.271,21.461,-42.142
C07076=1017.536,61.596,-125.666,-24.270,21.462,-42.146
C07077=1017.539,61.196,-125.630,-24.270,21.462,-42.150
C07078=1017.542,60.796,-125.593,-24.269,21.462,-42.155
C07079=1017.545,60.396,-125.557,-24.269,21.463,-42.159
C07080=1017.548,59.996,-125.521,-24.268,21.463,-42.163
C07081=1017.550,59.596,-125.485,-24.268,21.464,-42.166
C07082=1017.554,59.195,-125.449,-24.267,21.463,-42.172
C07083=1017.558,58.795,-125.412,-24.266,21.464,-42.175
C07084=1017.561,58.395,-125.376,-24.266,21.464,-42.179
C07085=1017.563,57.995,-125.340,-24.265,21.465,-42.183
C07086=1017.566,57.595,-125.304,-24.264,21.465,-42.188
C07087=1017.569,57.195,-125.268,-24.264,21.465,-42.192
C07088=1017.572,56.794,-125.231,-24.264,21.466,-42.196
C07089=1017.575,56.394,-125.196,-24.263,21.465,-42.201
C07090=1017.578,55.993,-125.159,-24.262,21.467,-42.205
C07091=1017.581,55.593,-125.123,-24.262,21.467,-42.209
C07092=1017.583,55.194,-125.088,-24.261,21.468,-42.212
C07093=1017.585,54.793,-125.051,-24.260,21.468,-42.218
C07094=1017.588,54.393,-125.015,-24.260,21.468,-42.221
C07095=1017.592,53.993,-124.980,-24.259,21.468,-42.225
C07096=1017.594,53.592,-124.943,-24.259,21.468,-42.230
C07097=1017.597,53.193,-124.907,-24.258,21.469,-42.234
C07098=1017.600,52.793,-124.871,-24.258,21.469,-42.238
C07099=1017.602,52.393,-124.835,-24.257,21.469,-42.243
C07100=1017.606,51.992,-124.800,-24.256,21.470,-42.247
C07101=1017.608,51.591,-124.763,-24.256,21.471,-42.251
C07102=1017.610,51.192,-124.728,-24.255,21.471,-42.255
C07103=1017.613,50.792,-124.691,-24.255,21.471,-42.260
C07104=1017.616,50.392,-124.655,-24.254,21.472,-42.264
C07105=1017.618,49.991,-124.620,-24.254,21.472,-42.268
C07106=1017.622,49.592,-124.584,-24.253,21.472,-42.273
C07107=1017.624,49.191,-124.548,-24.252,21.473,-42.277
C07108=1017.626,48.791,-124.512,-24.251,21.472,-42.282
C07109=1017.629,48.390,-124.476,-24.251,21.474,-42.286
C07110=1017.631,47.991,-124.441,-24.251,21.474,-42.290
C07111=1017.635,47.591,-124.405,-24.250,21.474,-42.295
C07112=1017.636,47.191,-124.369,-24.249,21.475,-42.299
C07113=1017.640,46.790,-124.333,-24.249,21.475,-42.302
C07114=1017.641,46.390,-124.297,-24.248,21.475,-42.308
C07115=1017.644,45.990,-124.262,-24.247,21.475,-42.311
C07116=1017.647,45.591,-124.226,-24.247,21.477,-42.316
C07117=1017.648,45.190,-124.190,-24.246,21.477,-42.321
C07118=1017.651,44.790,-124.155,-24.246,21.477,-42.325
C07119=1017.654,44.390,-124.119,-24.245,21.477,-42.330
C07120=1017.656,43.990,-124.083,-24.244,21.477,-42.333
C07121=1017.658,43.591,-124.048,-24.244,21.479,-42.338
C07122=1017.661,43.189,-124.012,-24.243,21.479,-42.343
C07123=1017.663,42.790,-123.976,-24.243,21.479,-42.347
C07124=1017.666,42.390,-123.941,-24.242,21.479,-42.352
C07125=1017.667,41.990,-123.905,-24.241,21.479,-42.356
C07126=1017.670,41.590,-123.870,-24.241,21.480,-42.359
C07127=1017.672,41.190,-123.834,-24.240,21.481,-42.365
C07128=1017.674,40.790,-123.799,-24.240,21.481,-42.369
C07129=1017.677,40.390,-123.762,-24.239,21.481,-42.374
C07130=1017.680,39.990,-123.728,-24.238,21.481,-42.378
C07131=1017.681,39.590,-123.692,-24.238,21.482,-42.383
C07132=1017.684,39.190,-123.656,-24.237,21.483,-42.387
C07133=1017.686,38.791,-123.621,-24.237,21.483,-42.391
C07134=1017.687,38.390,-123.586,-24.236,21.483,-42.396
C07135=1017.690,37.991,-123.551,-24.235,21.483,-42.400
C07136=1017.692,37.591,-123.515,-24.235,21.484,-42.405
C07137=1017.694,37.191,-123.479,-24.234,21.485,-42.409
C07138=1017.696,36.791,-123.444,-24.233,21.484,-42.414
C07139=1017.699,36.391,-123.409,-24.233,21.485,-42.418
C07140=1017.701,35.992,-123.373,-24.232,21.486,-42.424
C07141=1017.702,35.592,-123.338,-24.231,21.486,-42.428
C07142=1017.704,35.192,-123.303,-24.231,21.486,-42.433
C07143=1017.707,34.792,-123.268,-24.230,21.486,-42.437
C07144=1017.709,34.393,-123.233,-24.229,21.487,-42.442
C07145=1017.710,33.993,-123.197,-24.229,21.488,-42.446
C07146=1017.713,33.593,-123.161,-24.228,21.487,-42.451
C07147=1017.714,33.194,-123.126,-24.228,21.489,-42.455
C07148=1017.717,32.794,-123.092,-24.227,21.489,-42.461
C07149=1017.718,32.394,-123.057,-24.226,21.489,-42.464
C07150=1017.720,31.994,-123.021,-24.226,21.489,-42.469
C07151=1017.722,31.595,-122.986,-24.225,21.490,-42.474
C07152=1017.724,31.196,-122.950,-24.224,21.490,-42.479
C07153=1017.726,30.796,-122.916,-24.224,21.491,-42.483
C07154=1017.728,30.396,-122.881,-24.223,21.491,-42.488
C07155=1017.730,29.997,-122.846,-24.223,21.492,-42.492
C07156=1017.731,29.597,-122.810,-24.222,21.492,-42.497
C07157=1017.733,29.197,-122.775,-24.221,21.492,-42.501
C07158=1017.735,28.798,-122.741,-24.221,21.493,-42.507
C07159=1017.737,28.398,-122.706,-24.220,21.493,-42.510
C07160=1017.738,27.999,-122.671,-24.219,21.493,-42.516
C07161=1017.740,27.600,-122.636,-24.219,21.495,-42.520
C07162=1017.742,27.200,-122.600,-24.218,21.494,-42.525
C07163=1017.744,26.801,-122.565,-24.218,21.495,-42.529
C07164=1017.745,26.402,-122.530,-24.217,21.496,-42.534
C07165=1017.747,26.002,-122.496,-24.216,21.496,-42.540
C07166=1017.749,25.603,-122.461,-24.215,21.496,-42.543
C07167=1017.750,25.204,-122.426,-24.215,21.497,-42.549
